// 等待機械復位完成
IF NOT xExecute THEN
	IF Cylinder.List.fbSameSizeCV_Block2.InRearPosition AND
	   Cylinder.List.fbTransmitCV_CamaraHoriz.InRearPosition AND
	   Motor.List.TransmitSameSideCV.InStopped THEN
		xComplete := TRUE;
	END_IF
ELSE
	IF Motor.List.TransmitSameSideCV.InStopped THEN
		xComplete := TRUE;
	END_IF
END_IF
END_METHOD

METHOD CyclicAction
VAR_INPUT
    itfTimingController : CBML.ITimingController;
END_VAR
VAR_OUTPUT
    xComplete : BOOL := TRUE;
    iErrorID : INT := 0;
END_VAR
VAR_INST
	bMoveConveyorBackward:BOOL;
END_VAR
xComplete := FALSE;
// Phase 2:寫請求,由 FB_MachineControl.A20_ConveyorArbitration 驅動 motor
IF __ISVALIDREF(SameSizeCVRequest) THEN
	SameSizeCVRequest.bCamera_NeedBackward := bMoveConveyorBackward;
END_IF

CASE uiCyclicStep OF
	0:	// 初始化
		bMoveConveyorBackward:=FALSE;
		uiCyclicStep :=1000;

	1000:	// 擋盒子 (Block2)
		TON_TimeOut.IN:=TRUE;
		Cylinder.List.fbSameSizeCV_Block2.M_Extend();
		Cylinder.List.fbTransmitCV_CamaraHoriz.M_Retract();
		IF Cylinder.List.fbSameSizeCV_Block2.InFrontPosition AND
			Cylinder.List.fbTransmitCV_CamaraHoriz.InRearPosition THEN
			TON_TimeOut.IN:=FALSE;
			uiCyclicStep :=1050;
		END_IF
		IF TON_TimeOut.Q THEN
			uiResumeStep := uiCyclicStep;
			iErrorID := 10;
		END_IF

	1050:	// 馬達反轉
		TON_ConveyorTimeOut.IN:=TRUE;
		bMoveConveyorBackward:=TRUE;
		Cylinder.List.fbSameSizeCV_Press1.M_Retract();
		IF Motor.List.TransmitSameSideCV.InBackWard AND
			Cylinder.List.fbSameSizeCV_Press1.InRearPosition THEN
			TON_ConveyorTimeOut.IN:= FALSE;
			uiCyclicStep :=1100;
		END_IF
		IF TON_ConveyorTimeOut.Q THEN
			uiResumeStep := uiCyclicStep;
			iErrorID := 10;
		END_IF

	1100:	// 檢查盒子到達擋塊 (Phase 2:撤銷 backward + 請求 HoldStill 拍照位)
		TON_ArriviedTimeOut.IN:=TRUE;
		TON_DelaySensor.IN:=Input.bSameSizeCV_BoxDetect2_Sensor;
		IF TON_DelaySensor.Q THEN
			TON_DelaySensor.IN :=FALSE;
			TON_ArriviedTimeOut.IN :=FALSE;
			Cylinder.List.fbSameSizeCV_Press1.M_Extend();
			bMoveConveyorBackward:=FALSE;
			IF __ISVALIDREF(SameSizeCVRequest) THEN
				SameSizeCVRequest.bCamera_NeedBackward := FALSE;
				SameSizeCVRequest.bCamera_HoldStill    := TRUE;	// 拍照位必須靜止
			END_IF
			uiCyclicStep :=1200;
		END_IF
		IF TON_ArriviedTimeOut.Q THEN
			uiResumeStep := uiCyclicStep;
			iErrorID := 9;
		END_IF

	1200:	// 發送拍照請求 & 壓住盒子
		TON_ConveyorTimeOut.IN:=TRUE;
		IF Cylinder.List.fbSameSizeCV_Press1.InFrontPosition AND
			Motor.List.TransmitSameSideCV.InStopped THEN
			TON_ConveyorTimeOut.IN:= FALSE;
			UseBoxCamera :=TRUE;
			uiCyclicStep :=1300;
		END_IF
		IF TON_ConveyorTimeOut.Q THEN
			uiResumeStep := uiCyclicStep;
			iErrorID := 10;
		END_IF

	1300:	// 等待 C# 拍照完成 (Camera 錯誤不可續做) — Phase 2:解 HoldStill,再次請求 backward
		TON_CameraTimeOut.IN:=TRUE;
		IF BoxCameraDone THEN
			TON_CameraTimeOut.IN :=FALSE;
			Cylinder.List.fbSameSizeCV_Block2.M_Retract();
			bMoveConveyorBackward:=TRUE;
			IF __ISVALIDREF(SameSizeCVRequest) THEN
				SameSizeCVRequest.bCamera_HoldStill := FALSE;
			END_IF
			uiCyclicStep :=1400;
		END_IF
		IF TON_CameraTimeOut.Q THEN
			uiResumeStep := uiCyclicStep;
			iErrorID := 11;
		END_IF

	1400:	// 盒子通過 Detect1 感測器
		TON_TimeOut.IN :=TRUE;
		IF Input.bSameSizeCV_BoxDetect3_Sensor THEN
			TON_TimeOut.IN :=FALSE;
			uiCyclicStep :=1500;
		END_IF
		IF TON_TimeOut.Q THEN
			uiResumeStep := uiCyclicStep;
			iErrorID := 12;
		END_IF

	1500:	// 離開感測器後撤銷 backward (Phase 2:arbiter 自動停)
		TON_DelaySensor.IN :=TRUE;
		IF NOT Input.bSameSizeCV_BoxDetect3_Sensor THEN
			TON_DelaySensor.IN :=FALSE;
			bMoveConveyorBackward:=FALSE;
			IF __ISVALIDREF(SameSizeCVRequest) THEN
				SameSizeCVRequest.bCamera_NeedBackward := FALSE;
			END_IF
			uiCyclicStep :=1600;
		END_IF
		IF TON_DelaySensor.Q THEN
			TON_DelaySensor.IN:=FALSE;
			bMoveConveyorBackward:=FALSE;
			IF __ISVALIDREF(SameSizeCVRequest) THEN
				SameSizeCVRequest.bCamera_NeedBackward := FALSE;
			END_IF
			uiCyclicStep :=1600;
		END_IF

	1600:	// 等待馬達停止
		IF Motor.List.TransmitSameSideCV.InStopped THEN
			xComplete :=TRUE;
		END_IF

END_CASE

IF TON_SameSizeBoxDetect1_Delay.Q THEN
	iErrorID := 13;
END_IF
END_METHOD

METHOD ExitAction
VAR_INPUT
    xAfterCleanup : BOOL;
    xInCopyCode : BOOL;
END_VAR
	uiCyclicStep    := 0;
	xAfterCleanup := true;
END_METHOD

METHOD M_GetErrorMsg : T_MaxString
VAR_INPUT
	xErrorID: INT;
END_VAR

VAR

END_VAR
CASE xErrorID OF
	1:
		M_GetErrorMsg := 'No Error';
	2:
		M_GetErrorMsg := 'FB_SameSizeCVCamera_Reverse ErrorID 2: Action time out';
	3:
		M_GetErrorMsg := 'FB_SameSizeCVCamera_Reverse ErrorID 3: Position Data invalid';
	4:
		M_GetErrorMsg := 'FB_SameSizeCVCamera_Reverse ErrorID 4: Block1 cylinder not ready';
	5:
		M_GetErrorMsg := 'FB_SameSizeCVCamera_Reverse ErrorID 5: Block2 cylinder not ready';
	6:
		M_GetErrorMsg := 'FB_SameSizeCVCamera_Reverse ErrorID 6: Press1 cylinder not ready';
	7:
		M_GetErrorMsg := 'FB_SameSizeCVCamera_Reverse ErrorID 7: Press2 cylinder not ready';
	8:
		M_GetErrorMsg := 'FB_SameSizeCVCamera_Reverse ErrorID 8: CameraHoriz cylinder not ready';
	9:
		M_GetErrorMsg :='FB_SameSizeCVCamera_Reverse ErrorID 9:  Box not arrived ';
	10:
		M_GetErrorMsg :='FB_SameSizeCVCamera_Reverse ErrorID 10: Cylinder timeout';
	11:
		M_GetErrorMsg :='FB_SameSizeCVCamera_Reverse ErrorID 11: C# BoxCameraDone timeout';
	12:
		M_GetErrorMsg :='FB_SameSizeCVCamera_Reverse ErrorID 12: Box cross sensor timeout';
	13:
		M_GetErrorMsg :='FB_SameSizeCVCamera_Reverse ErrorID 13: SameSizeConveyor full box infront ';
END_CASE
END_METHOD

METHOD ResetAction
VAR_OUTPUT
    xComplete : BOOL := TRUE;
END_VAR
xComplete := FALSE;

// ============================================================
// Resume 機制判斷
// ------------------------------------------------------------
// 當錯誤發生後，操作員可選擇：
//   1. 保持 xExecute = TRUE 並按 Reset → Resume (從錯誤點繼續)
//   2. 先關閉 xExecute，再重新啟動 → 從頭開始
// ============================================================
bResumeEnabled := xExecute;

// 如果不是 Resume 模式，清除 Resume 步驟記錄
IF NOT bResumeEnabled THEN
	uiResumeStep := 0;
END_IF

// 清除所有 Timer
TON_DelaySensor.IN 		:= FALSE;
TON_TimeOut.IN 			:= FALSE;
TON_ArriviedTimeOut.IN 	:= FALSE;
TON_CameraTimeOut.IN 	:= FALSE;
TON_ConveyorTimeOut.IN 	:= FALSE;

xComplete := TRUE;
END_METHOD

METHOD StartAction
VAR_OUTPUT
    xComplete : BOOL := TRUE;
	iErrorID : INT := 0;
END_VAR
VAR
	bIsResumeMode : BOOL;	// 局部變數：記錄是否為 Resume 模式
END_VAR
xComplete := FALSE;

// 清除所有 Timer
TON_DelaySensor.IN 		:= FALSE;
TON_TimeOut.IN 			:= FALSE;
TON_ArriviedTimeOut.IN 	:= FALSE;
TON_CameraTimeOut.IN 	:= FALSE;
TON_ConveyorTimeOut.IN 	:= FALSE;

// ============================================================
// Resume 機制處理
// ------------------------------------------------------------
// 可 Resume 的錯誤: 氣缸/馬達/等待盒子
// 不可 Resume 的錯誤: Step 1300 (C# 拍照失敗)
// ============================================================
bIsResumeMode := bResumeEnabled AND uiResumeStep > 0 AND uiResumeStep <> 1300;

IF bResumeEnabled AND uiResumeStep > 0 THEN
	IF uiResumeStep = 1300 THEN
		// Camera 錯誤：不可 Resume，強制從頭開始
		uiCyclicStep 	:= 0;
		UseBoxCamera 	:= FALSE;
		BoxCameraDone 	:= FALSE;
	ELSE
		// 其他錯誤：允許 Resume (人工已確認可繼續)
		uiCyclicStep := uiResumeStep;
	END_IF
	// 清除 Resume 旗標
	bResumeEnabled 	:= FALSE;
	uiResumeStep 	:= 0;
ELSE
	// 正常模式：從頭開始
	uiCyclicStep 	:= 0;
	UseBoxCamera 	:= FALSE;
	BoxCameraDone 	:= FALSE;
END_IF

// ============================================================
// 啟動前錯誤檢查
// ============================================================
IF TON_SameSizeBoxDetect1_Delay.Q THEN
	iErrorID := 13;
END_IF

IF Cylinder.List.fbSameSizeCV_Block1.xError THEN
	iErrorID := 4;
END_IF
IF Cylinder.List.fbSameSizeCV_Block2.xError THEN
	iErrorID := 5;
END_IF
IF Cylinder.List.fbSameSizeCV_Press1.xError THEN
	iErrorID := 6;
END_IF
IF Cylinder.List.fbSameSizeCV_Press2.xError THEN
	iErrorID := 7;
END_IF
IF Cylinder.List.fbTransmitCV_CamaraHoriz.xError THEN
	iErrorID := 8;
END_IF
IF Motor.List.TransmitSameSideCV.xError THEN
	iErrorID := 9;
END_IF

// 完成條件：Resume 模式直接完成，正常模式需檢查初始位置
IF bIsResumeMode OR
   (Cylinder.List.fbSameSizeCV_Block2.InRearPosition AND
    Motor.List.TransmitSameSideCV.InStopped) THEN
	xComplete := TRUE;
END_IF
END_METHOD

END_FUNCTION_BLOCK

// ---- Library/20_MachineUnits/22_AllocateArea/Service/FB_DifferentCVCamera.TcPOU
FUNCTION_BLOCK FB_DifferentCVCamera EXTENDS FB_ActionBasic
VAR_INPUT
    xExecute    : BOOL;
    xAbort      : BOOL;
	xReset		: BOOL;
    Cylinder 	: REFERENCE TO UNI_CylinderList;
    TimeOut  	: LREAL := 600; // Unit : s
	Input		: ST_InputTable;
	OutPut		: ST_OutputTable;
	Motor		: REFERENCE TO UNI_MotorList;
	BoxCameraDone :BOOL;
END_VAR	
VAR_OUTPUT
    xAborted : BOOL;
    iErrorID : INT;
    ErrorMsg : STRING;
	UseBoxCamera	:BOOL;
END_VAR
VAR
    StateBehaviour   : CBML.ETrigATo;
    CurrentPosition : ST_PositionTable;
	uiCyclicStep    : UINT := 0;
	TON_DelaySensor	:TON;
	TON_TimeOut		:TON;
	TON_ArriviedTimeOut :TON ;
	TON_CameraTimeOut	:TON;
	TON_ConveyorTimeOut	:TON;
	Reset_Rtrig 	:R_TRIG;
	fbExecuteEdgeDetect :FB_EdgeDetect;
	// ========== Resume 續做機制 ==========
	uiResumeStep	: UINT := 0;		// 錯誤發生時記錄的步驟，供續做使用
	bResumeEnabled	: BOOL := FALSE;	// 續做模式啟用旗標
END_VAR

THIS^.IBehaviourModel := StateBehaviour;
StateBehaviour(xExecute := xExecute,
              xAbort := xAbort OR fbExecuteEdgeDetect.xFallingEdge,
              udiTimeOut := LREAL_TO_UDINT( TimeOut*1000000),
              xDone => xDone,
              xBusy => xBusy,
              xError => xError,
              xAborted => xAborted);

iErrorID := StateBehaviour._model.iErrorID;
ErrorMsg := M_GetErrorMsg(xErrorID := iErrorID);

fbExecuteEdgeDetect(xInput :=xExecute);

Reset_Rtrig(CLK:= xReset);
IF Reset_Rtrig.Q THEN
	StateBehaviour.ResetModel(xCommit:=xReset);
END_IF

A00_BaseUnits();

ACTION A00_BaseUnits:
TON_DelaySensor(PT:= T#1S);
TON_TimeOut(PT := T#20S);
TON_ArriviedTimeOut(PT:= T#60S);
TON_CameraTimeOut(PT :=T#250S);
TON_ConveyorTimeOut(PT :=T#60S);
END_ACTION

METHOD CleanupAction
VAR_INPUT
    xAbortProposed : BOOL;
    iErrorIDProposed: INT;
END_VAR
VAR_OUTPUT
    xComplete : BOOL := TRUE;
    xAbort: BOOL := xAbortProposed;
 	iErrorID : INT := iErrorIDProposed;
END_VAR
xComplete := FALSE;

// ============================================================
// Resume 機制：保存當前步驟供後續 Resume 使用
// ============================================================
IF uiResumeStep = 0 THEN
	uiResumeStep := uiCyclicStep;
END_IF

// 清除所有 Timer
TON_DelaySensor.IN 		:= FALSE;
TON_TimeOut.IN 			:= FALSE;
TON_ArriviedTimeOut.IN 	:= FALSE;
TON_CameraTimeOut.IN 	:= FALSE;
TON_ConveyorTimeOut.IN 	:= FALSE;

// 重置輸出信號
UseBoxCamera 	:= FALSE;
BoxCameraDone 	:= FALSE;

// 機械復位到安全狀態
IF NOT xExecute THEN 
	Cylinder.List.fbDifferentSizeCV_Block1.M_Retract();
END_IF
Motor.List.TransmitDifferentSideCV.M_MotorStop();

// 等待機械復位完成
IF NOT xExecute THEN
	IF Cylinder.List.fbDifferentSizeCV_Block1.InRearPosition AND
	   Motor.List.TransmitDifferentSideCV.InStopped THEN
		xComplete := TRUE;
	END_IF
ELSE	
	IF Motor.List.TransmitDifferentSideCV.InStopped THEN
		xComplete := TRUE;
	END_IF
END_IF
END_METHOD

METHOD CyclicAction
VAR_INPUT
    itfTimingController : CBML.ITimingController;
END_VAR
VAR_OUTPUT
    xComplete : BOOL := TRUE;
    iErrorID : INT := 0;
END_VAR
VAR_INST
	bMoveConveyorForward	 : BOOL;
END_VAR
xComplete := FALSE;
IF bMoveConveyorForward THEN
	IF NOT Motor.List.TransmitDifferentSideCV.InBackWard THEN
		Motor.List.TransmitDifferentSideCV.M_MoveForward();
	END_IF
END_IF
CASE uiCyclicStep OF
	0:	// 初始化
		bMoveConveyorForward:=FALSE;
		uiCyclicStep :=1000;
		
	1000:	// 擋第一個盒子
		TON_TimeOut.IN:=TRUE;
		Cylinder.List.fbDifferentSizeCV_Block1.M_Extend();
		Cylinder.List.fbTransmitCV_CamaraHoriz.M_Extend();
		IF Cylinder.List.fbDifferentSizeCV_Block1.InFrontPosition AND
			Cylinder.List.fbTransmitCV_CamaraHoriz.InFrontPosition THEN
			TON_TimeOut.IN:=FALSE;
			uiCyclicStep :=1050;
		END_IF
		IF TON_TimeOut.Q THEN
			uiResumeStep := uiCyclicStep;
			iErrorID := 7;
		END_IF

	1050:	// 馬達前進
		TON_ConveyorTimeOut.IN:=TRUE;
		bMoveConveyorForward:=TRUE;
		Cylinder.List.fbDifferentSizeCV_Press1.M_Retract();
		IF Motor.List.TransmitDifferentSideCV.InForWard AND
			Cylinder.List.fbDifferentSizeCV_Press1.InRearPosition THEN
			TON_ConveyorTimeOut.IN:= FALSE;
			uiCyclicStep :=1100;
		END_IF
		IF TON_ConveyorTimeOut.Q THEN
			uiResumeStep := uiCyclicStep;
			iErrorID := 7;
		END_IF

	1100:	// 檢查盒子到達擋塊
		TON_ArriviedTimeOut.IN:=TRUE;
		TON_DelaySensor.IN:=Input.bDifferentSizeCV_BoxDetect2_Sensor;
		IF TON_DelaySensor.Q THEN
			TON_DelaySensor.IN :=FALSE;
			TON_ArriviedTimeOut.IN :=FALSE;
			Cylinder.List.fbDifferentSizeCV_Press1.M_Extend();
			bMoveConveyorForward:=FALSE;
			Motor.List.TransmitDifferentSideCV.M_MotorStop();
			uiCyclicStep :=1200;
		END_IF
		IF TON_ArriviedTimeOut.Q THEN
			uiResumeStep := uiCyclicStep;
			iErrorID := 8;
		END_IF

	1200:	// 發送拍照請求 & 擋住第二個盒子
		TON_ConveyorTimeOut.IN:=TRUE;
		IF Cylinder.List.fbDifferentSizeCV_Press1.InFrontPosition AND
			Motor.List.TransmitDifferentSideCV.InStopped THEN
			TON_ConveyorTimeOut.IN:= FALSE;
			UseBoxCamera :=TRUE;
			uiCyclicStep :=1300;
		END_IF
		IF TON_ConveyorTimeOut.Q THEN
			uiResumeStep := uiCyclicStep;
			iErrorID := 9;
		END_IF

	1300:	// 等待 C# 拍照完成 (Camera 錯誤不可續做)
		TON_CameraTimeOut.IN:=TRUE;
		IF BoxCameraDone THEN
			TON_CameraTimeOut.IN :=FALSE;
			Cylinder.List.fbDifferentSizeCV_Block1.M_Retract();
			bMoveConveyorForward:=TRUE;
			uiCyclicStep :=1400;
		END_IF
		IF TON_CameraTimeOut.Q THEN
			uiResumeStep := uiCyclicStep;
			iErrorID :=10;
		END_IF

	1400:	// 盒子通過 Detect1 感測器
		TON_TimeOut.IN :=TRUE;
		IF Input.bDifferentSizeCV_BoxDetect1_Sensor THEN
			TON_TimeOut.IN :=FALSE;
			uiCyclicStep :=1500;
		END_IF
		IF TON_TimeOut.Q THEN
			uiResumeStep := uiCyclicStep;
			iErrorID :=11;
		END_IF

	1500:	// 離開感測器後停止馬達
		TON_DelaySensor.IN:=TRUE;
		IF NOT Input.bDifferentSizeCV_BoxDetect1_Sensor THEN
			TON_DelaySensor.IN:=FALSE;
			bMoveConveyorForward:=FALSE;
			Motor.List.TransmitDifferentSideCV.M_MotorStop();
			uiCyclicStep :=1600;
		END_IF
		IF TON_DelaySensor.Q THEN
			TON_DelaySensor.IN:=FALSE;
			bMoveConveyorForward:=FALSE;
			Motor.List.TransmitDifferentSideCV.M_MotorStop();
			uiCyclicStep :=1600;
		END_IF
	
	1600:	// 等待馬達停止
		IF Motor.List.TransmitDifferentSideCV.InStopped THEN
			xComplete :=TRUE;
		END_IF

END_CASE
END_METHOD

METHOD ExitAction
VAR_INPUT
    xAfterCleanup : BOOL;
    xInCopyCode : BOOL;
END_VAR
END_METHOD

METHOD M_GetErrorMsg : T_MaxString
VAR_INPUT
	xErrorID: INT;
END_VAR

VAR
	
END_VAR
CASE xErrorID OF
	0:
		M_GetErrorMsg := 'No Error';
	1:
		M_GetErrorMsg := 'FB_DifferentCVCamera ErrorID 1: Action time out';
	2:
		M_GetErrorMsg := 'FB_DifferentCVCamera ErrorID 2: Position Data invalid';
	3:
		M_GetErrorMsg := 'FB_DifferentCVCamera ErrorID 3: Block1 cylinder not ready';
	4:
		M_GetErrorMsg := 'FB_DifferentCVCamera ErrorID 4: Press1 cylinder not ready';
	5:
		M_GetErrorMsg := 'FB_DifferentCVCamera ErrorID 5: CamaraHoriz cylinder not ready';
	6:
		M_GetErrorMsg := 'FB_DifferentCVCamera ErrorID 6: DifferentCV not ready ';
	7:
		M_GetErrorMsg := 'FB_DifferentCVCamera ErrorID 7: Cylinder timeout';
	8:
		M_GetErrorMsg :='FB_DifferentCVCamera ErrorID 8: photo area have not box timeout';
	9:
		M_GetErrorMsg :='FB_DifferentCVCamera ErrorID 9: motor & cylinder timeout';
	10:
		M_GetErrorMsg :='FB_DifferentCVCamera ErrorID 10: C# BoxCameraDone timeout';
	11:
		M_GetErrorMsg :='FB_DifferentCVCamera ErrorID 11: Box cross sensor not detact timeout';
		
	20:
		M_GetErrorMsg :='FB_DifferentCVCamera ErrorID 20: Differnet conveyor full box infront';
END_CASE
END_METHOD

METHOD ResetAction
VAR_OUTPUT
    xComplete : BOOL := TRUE;
END_VAR
xComplete := FALSE;

// ============================================================
// Resume 機制判斷
// ------------------------------------------------------------
// 當錯誤發生後，操作員可選擇：
//   1. 保持 xExecute = TRUE 並按 Reset → Resume (從錯誤點繼續)
//   2. 先關閉 xExecute，再重新啟動 → 從頭開始
// ============================================================
bResumeEnabled := xExecute;

// 如果不是 Resume 模式，清除 Resume 步驟記錄
IF NOT bResumeEnabled THEN
	uiResumeStep := 0;
END_IF

// 清除所有 Timer
TON_DelaySensor.IN 		:= FALSE;
TON_TimeOut.IN 			:= FALSE;
TON_ArriviedTimeOut.IN 	:= FALSE;
TON_CameraTimeOut.IN 	:= FALSE;
TON_ConveyorTimeOut.IN 	:= FALSE;

xComplete := TRUE;
END_METHOD

METHOD StartAction
VAR_OUTPUT
    xComplete : BOOL := TRUE;
	iErrorID : INT := 0;
END_VAR
VAR
	bIsResumeMode : BOOL;	// 局部變數：記錄是否為 Resume 模式
END_VAR
xComplete := FALSE;

// 清除所有 Timer
TON_DelaySensor.IN 		:= FALSE;
TON_TimeOut.IN 			:= FALSE;
TON_ArriviedTimeOut.IN 	:= FALSE;
TON_CameraTimeOut.IN 	:= FALSE;
TON_ConveyorTimeOut.IN 	:= FALSE;

// ============================================================
// Resume 機制處理
// ------------------------------------------------------------
// 可 Resume 的錯誤: Error 7, 8, 9, 11 (氣缸/馬達/等待盒子)
// 不可 Resume 的錯誤: Error 10 (C# 拍照失敗), Error 20 (輸送帶滿載)
// ============================================================
bIsResumeMode := bResumeEnabled AND uiResumeStep > 0 AND uiResumeStep <> 1300;

IF bResumeEnabled AND uiResumeStep > 0 THEN
	IF uiResumeStep = 1300 THEN
		// Camera 錯誤：不可 Resume，強制從頭開始
		uiCyclicStep 	:= 0;
		UseBoxCamera 	:= FALSE;
		BoxCameraDone 	:= FALSE;
	ELSE
		// 其他錯誤：允許 Resume (人工已確認可繼續)
		uiCyclicStep := uiResumeStep;
	END_IF
	// 清除 Resume 旗標
	bResumeEnabled 	:= FALSE;
	uiResumeStep 	:= 0;
ELSE
	// 正常模式：從頭開始
	uiCyclicStep 	:= 0;
	UseBoxCamera 	:= FALSE;
	BoxCameraDone 	:= FALSE;
END_IF

// ============================================================
// 啟動前錯誤檢查
// ============================================================
IF Input.bDifferentSizeCV_BoxDetect1_Sensor THEN
	iErrorID := 20;
END_IF

IF Cylinder.List.fbDifferentSizeCV_Block1.xError THEN
	iErrorID := 3;
END_IF
IF Cylinder.List.fbDifferentSizeCV_Press1.xError THEN
	iErrorID := 4;
END_IF
IF Cylinder.List.fbTransmitCV_CamaraHoriz.xError THEN
	iErrorID := 5;
END_IF
IF Motor.List.TransmitDifferentSideCV.xError THEN
	iErrorID := 6;
END_IF

// 完成條件：Resume 模式直接完成，正常模式需檢查初始位置
IF bIsResumeMode OR
   (Cylinder.List.fbDifferentSizeCV_Block1.InRearPosition AND
    Motor.List.TransmitDifferentSideCV.InStopped) THEN
	xComplete := TRUE;
END_IF
END_METHOD

END_FUNCTION_BLOCK

// ---- Library/20_MachineUnits/22_AllocateArea/Service/FB_SameSizeCV_ReverseBatchPickAndPhoto.TcPOU
// FB_SameSizeCV_ReverseBatchPickAndPhoto
// 逆向拍照批次入料服務
// Pipeline 三軌平行:
//   Track 1 (小手臂): 從鐵盤取盒放到同尺寸軌道 (ShippingRobotTransfer)
//   Track 2 (拍照):   觸發逆向拍照, 接收 C# 回傳結果
//   Track 3 (大手臂): 雙爪/單爪搬運到倉庫或 NG 區 (倉儲 Fanuc Robot)
//
// 狀態機架構: FB_ObjectBase_V2 + IBasicElement
//   DORMANT → EXECUTING → DONE / ABORTING → ABORTED → RESETTING → DORMANT
//
// Handshake: 由 FB_AllocateAreaWithRoundbelt 逐欄位 link ADS 結構

FUNCTION_BLOCK FB_SameSizeCV_ReverseBatchPickAndPhoto EXTENDS FB_ObjectBase_V2 IMPLEMENTS IBasicElement

VAR_INPUT
	// ===== 鐵盤 Sensor (C# → PLC, 目前 C# 模擬，後續改硬體訊號) =====
	bLeftPlateReady		: BOOL;
	bRightPlateReady	: BOOL;

	// ===== 鐵盤配置 (C# → PLC) =====
	LeftPlate			: ARRAY[0..3] OF BOOL;
	RightPlate			: ARRAY[0..3] OF BOOL;
	bLeftConfigReady	: BOOL;
	bRightConfigReady	: BOOL;

	// ===== 拍照結果 (C# → PLC) =====
	BoxCameraDone		: BOOL;
	CameraIsOK			: BOOL;
	CameraWarehouse		: INT;
	CameraLevel			: INT;
	CameraTrack			: INT;

	// ===== 硬體 REFERENCE =====
	Cylinder			: REFERENCE TO UNI_CylinderList;
	Motor				: REFERENCE TO UNI_MotorList;
	SameSizeCVRequest	: REFERENCE TO ST_SameSizeCVRequest;	// Phase 2 仲裁,傳到 3 個 sub-FB
	Input				: ST_InputTable;
	OutPut				: ST_OutputTable;
	StorageRobot		: REFERENCE TO FB_FanucRobot_Basic_V2;
	ShippingRobot		: REFERENCE TO FB_FanucRobot_Basic_V2;
	WareHouse			: REFERENCE TO FB_WareHouse;
	
	Stop				: BOOL;

	// ===== 設定 =====
	PlateWaitTimeout	: TIME := T#60S;
	WaitPairTimeout		: TIME := T#15S;
	BatchTimeout		: TIME := T#600S;
END_VAR

VAR_OUTPUT
	// ===== 鐵盤狀態 (PLC → C#) =====
	bLeftPlateArrived	: BOOL;
	bRightPlateArrived	: BOOL;
	bLeftPlateDone		: BOOL;
	bRightPlateDone		: BOOL;

	// ===== 拍照請求 (PLC → C#) =====
	UseBoxCamera		: BOOL;

	// ===== 狀態監控 (PLC → C#) =====
	uiUnphotographedCount	: UINT;
	uiTotalProcessed		: UINT;
	uiTransportedCount		: UINT;
	
	
END_VAR

VAR
	strStatus			: STRING;
	_UniqueErrorCode	: STRING;
	_bRetry				: BOOL;

	// ===== Track 1: 小手臂取盒 =====
	uiPickStep				: UINT := 0;
	uiCurrentSide			: UINT := 0;		// 0=Left, 1=Right
	uiCurrentSlot			: UINT := 0;		// 0..3
	bPickTrackDone			: BOOL;
	bLeftProcessed			: BOOL;
	bRightProcessed			: BOOL;
	bLeftPlateReady_Prev	: BOOL;
	bRightPlateReady_Prev	: BOOL;
	bLeftConfigLatched		: BOOL;
	bRightConfigLatched		: BOOL;
	bLeftConfigReady_Prev	: BOOL;
	bRightConfigReady_Prev	: BOOL;

	// ===== Track 2: 拍照 =====
	uiCameraStep			: UINT := 0;
	uiCameraRequestCount	: UINT := 0;

	// ===== Track 3: 大手臂搬運 =====
	uiTransportStep		: UINT := 0;
	BoxQueue			: ST_ReverseBatchBoxQueue;
	stGripA				: ST_ReverseBatchBoxResult;
	stGripB				: ST_ReverseBatchBoxResult;
	bUseDualGrip		: BOOL;
	bTransportBusy		: BOOL;

	// ===== Timers =====
	tonTimeOut				: TON;
	TON_PlateWaitTimeout	: TON;
	TON_PickupTimeout		: TON;
	TON_CameraTimeout		: TON;
	TON_ConfigTimeout		: TON;
	TON_WaitPairTimeout		: TON;
	TON_CameraClearTimeout	: TON;

	// ===== Resume =====
	uiResumePickStep		: UINT := 0;
	uiResumeCameraStep		: UINT := 0;
	uiResumeTransportStep	: UINT := 0;
	
	// 內部使用Service
	ShippingTransfer	: FB_ShippingRobotTransfer;
	BoxToWareHouse		: FB_SameSizeCV_ReverseBoxToWareHouse;
	_fbSameSizeCV_ReverseCamera	: FB_SameSizeCVCamera_Reverse;
END_VAR

SUPER^.A10_StateControl();
A00_BasicUnits();

ACTION A00_BasicUnits:
tonTimeOut(PT := BatchTimeout);
TON_PlateWaitTimeout(PT := PlateWaitTimeout);
TON_PickupTimeout(PT := T#60S);
TON_CameraTimeout(PT := T#600S);
TON_ConfigTimeout(PT := T#60S);
TON_WaitPairTimeout(PT := WaitPairTimeout);
TON_CameraClearTimeout(PT := T#30S);


ShippingTransfer(
	Execute:= , 
	Abort:= , 
	Reset:= , 
	Pause:= , 
	ObjectName:= , 
	Busy=> , 
	Done=> , 
	Aborted=> , 
	Error=> , 
	Paused=> , 
	ErrorID=> , 
	Status=> , 
	UniqueErrorCode=> , 
	Robot:= ShippingRobot,
	Info:= ,
	Stop:= Stop,
	Input:= INPUT,
	Output:= OUTPUT,
	Motor:= Motor,
	SameSizeCVRequest:= SameSizeCVRequest,
	Cylinder:= Cylinder,
	Buzz:= ,
	RedLamp:= , 
	bCompleteRequest:= , 
	fbShippingHomingBusy:= , 
	bTransCVInPosition_Left=> , 
	bTransCVInPosition_Right=> );
	
BoxToWareHouse(
	Execute:= , 
	Abort:= , 
	Reset:= , 
	Pause:= , 
	ObjectName:= , 
	Busy=> , 
	Done=> , 
	Aborted=> , 
	Error=> , 
	Paused=> , 
	ErrorID=> , 
	Status=> , 
	UniqueErrorCode=> , 
	bBoxA_Enable:= ,
	eBoxA_Destination:= ,
	iBoxA_Warehouse:= ,
	iBoxA_Level:= ,
	iBoxA_Track:= ,
	iBoxA_PullOutSide:= ,
	bBoxB_Enable:= ,
	eBoxB_Destination:= ,
	iBoxB_Warehouse:= ,
	iBoxB_Level:= ,
	iBoxB_Track:= ,
	iBoxB_PullOutSide:= ,
	NGAreaPosition:= ,
	PickupPosition:= ,
	Cylinder:= Cylinder,
	Motor:= Motor,
	SameSizeCVRequest:= SameSizeCVRequest,
	Input:= Input,
	OutPut:= OutPut,
	StorageRobot:= StorageRobot,
	WareHouse:= WareHouse,
	PullOutConveyor:= ,
	Stop:= Stop,
	bBoxA_Done=> ,
	bBoxB_Done=> );
	
_fbSameSizeCV_ReverseCamera(
	xDone=> , 
	xBusy=> , 
	xError=> , 
	xExecute:= , 
	xAbort:= , 
	xReset:= , 
	Cylinder:= Cylinder,
	TimeOut:= ,
	Input:= input,
	OutPut:= output,
	Motor:= Motor,
	SameSizeCVRequest:= SameSizeCVRequest,
	BoxCameraDone:= ,
	xAborted=> , 
	iErrorID=> , 
	ErrorMsg=> , 
	UseBoxCamera=> );
END_ACTION

METHOD M_GetErrorMsg : T_MaxString
VAR_INPUT
END_VAR
IF _UniqueErrorCode = 'E_PICKUP_TIMEOUT' THEN
	M_GetErrorMsg := 'FB_SameSizeCV_ReverseBatchPickAndPhoto: ShippingRobot pickup timeout';
ELSIF _UniqueErrorCode = 'E_BIGARM_TIMEOUT' THEN
	M_GetErrorMsg := 'FB_SameSizeCV_ReverseBatchPickAndPhoto: BigArm transport timeout';
ELSIF _UniqueErrorCode = 'E_CONVEYOR_FULL' THEN
	M_GetErrorMsg := 'FB_SameSizeCV_ReverseBatchPickAndPhoto: Conveyor full (queue overflow)';
ELSIF _UniqueErrorCode = 'E_CONFIG_TIMEOUT' THEN
	M_GetErrorMsg := 'FB_SameSizeCV_ReverseBatchPickAndPhoto: Waiting C# plate config timeout';
ELSIF _UniqueErrorCode = 'E_CAMERA_TIMEOUT' THEN
	M_GetErrorMsg := 'FB_SameSizeCV_ReverseBatchPickAndPhoto: Camera timeout';
ELSIF _UniqueErrorCode = 'E_CAMERA_CLEAR_TIMEOUT' THEN
	M_GetErrorMsg := 'FB_SameSizeCV_ReverseBatchPickAndPhoto: C# did not clear BoxCameraDone';
ELSIF _UniqueErrorCode = 'E_BATCH_TIMEOUT' THEN
	M_GetErrorMsg := 'FB_SameSizeCV_ReverseBatchPickAndPhoto: Batch global timeout';
ELSIF _UniqueErrorCode = '' THEN
	M_GetErrorMsg := 'No Error';
ELSE
	M_GetErrorMsg := _UniqueErrorCode;
END_IF
END_METHOD

// 已中止狀態 — 等待 Reset 信號，支援 Resume
METHOD M_STATE_ABORTED
VAR_INPUT
END_VAR
IF NOT _bRetry THEN
	Busy 			:= FALSE;
	Aborted 		:= TRUE;
	Error 			:= TRUE;
	Status 			:= strStatus;
	uiAbortingStep 	:= 0;
	_AbortCompleted := FALSE;
END_IF


IF reset THEN
	_bRetry := TRUE;
	Aborted := FALSE;
	Error 	:= FALSE;	
END_IF

IF NOT Execute THEN
	eState := STATE_RESETTING;
END_IF

// 等待外部 Reset → 恢復或重置
IF Execute
	AND _bRetry 
	AND NOT StorageRobot._DI1.Error 
	AND NOT ShippingRobot._DI1.Error 
	AND NOT StorageRobot.Halt
	AND NOT StorageRobot.Halt
THEN
	status := 'FB_SameSizeCV_ReverseBatchPickAndPhoto: Retry Complete';
	// 恢復三軌步驟
	uiPickStep := uiResumePickStep;
	uiCameraStep := uiResumeCameraStep;
	uiTransportStep := uiResumeTransportStep;
	uiResumePickStep := 0;
	uiResumeCameraStep := 0;
	uiResumeTransportStep := 0;
	// 跳過初始化，直接進入三軌運行
	uiExecutingStep := 100;

	eState := STATE_RESETTING;
END_IF
END_METHOD

// 中止狀態 — 停止所有 Track，保存 Resume 步驟
METHOD M_STATE_ABORTING
VAR_INPUT
END_VAR
CASE uiAbortingStep OF
0:
	// 保存所有 Track Resume 步驟 (如果尚未保存)
	IF uiResumePickStep = 0 AND uiResumeTransportStep = 0 AND uiResumeCameraStep = 0 THEN
		uiResumePickStep := uiPickStep;
		uiResumeCameraStep := uiCameraStep;
		uiResumeTransportStep := uiTransportStep;
	END_IF

	// 清除所有 Timer
	tonTimeOut.IN				:= FALSE;
	TON_PlateWaitTimeout.IN		:= FALSE;
	TON_PickupTimeout.IN		:= FALSE;
	TON_CameraTimeout.IN		:= FALSE;
	TON_ConfigTimeout.IN		:= FALSE;
	TON_WaitPairTimeout.IN		:= FALSE;
	TON_CameraClearTimeout.IN	:= FALSE;

	// 清除輸出
	UseBoxCamera := FALSE;

	// 停止小手臂
	ShippingTransfer.Execute := FALSE;
	ShippingTransfer.Abort := TRUE;

	// 停止大手臂子服務
	BoxToWareHouse.Execute := FALSE;
	BoxToWareHouse.Abort := TRUE;

	uiAbortingStep := 100;

100:
	// 等待子服務停止 (ShippingTransfer + BoxToWareHouse)
	IF (NOT ShippingTransfer.Busy OR ShippingTransfer.Aborted)
	   AND (NOT BoxToWareHouse.Busy OR BoxToWareHouse.Aborted) THEN
		ShippingTransfer.Abort := FALSE;
		BoxToWareHouse.Abort := FALSE;
		uiAbortingStep := 9999;
	END_IF

9999:
	_AbortCompleted := TRUE;
END_CASE

IF NOT Execute THEN
	eState := STATE_RESETTING;
ELSIF _AbortCompleted THEN
	eState := STATE_Aborted;
END_IF
END_METHOD

METHOD M_STATE_DONE
VAR_INPUT
END_VAR
Busy := FALSE;
Done := TRUE;
tonTimeOut.IN := FALSE;

// 等待外部取消 Execute 後進入 RESETTING
IF NOT Execute THEN
	eState := STATE_RESETTING;
END_IF
END_METHOD

METHOD M_STATE_DORMANT
VAR_INPUT
END_VAR
VAR
	i : UINT;
END_VAR
// 清除所有輸出與內部狀態
Busy				:= FALSE;
Done				:= FALSE;
Aborted				:= FALSE;
Error				:= FALSE;
ErrorID				:= 0;
Status				:= '';
_ResetCompleted		:= FALSE;
_Error				:= FALSE;
_Executed			:= FALSE;
_Abort				:= FALSE;
uiExecutingStep		:= 0;
uiResettingStep		:= 0;
uiAbortingStep		:= 0;

tonTimeOut.IN		:= FALSE;
_UniqueErrorCode	:= '';
_bRetry				:= FALSE;

// 清除 Track 變數
uiPickStep 			:= 0;
uiCameraStep 		:= 0;
uiTransportStep 	:= 0;
uiCameraRequestCount := 0;
uiUnphotographedCount := 0;
uiTotalProcessed 	:= 0;
uiTransportedCount 	:= 0;
bPickTrackDone 		:= FALSE;
bLeftProcessed 		:= FALSE;
bRightProcessed 	:= FALSE;
bTransportBusy 		:= FALSE;
bUseDualGrip 		:= FALSE;
UseBoxCamera 		:= FALSE;
bLeftPlateArrived 	:= FALSE;
bRightPlateArrived 	:= FALSE;
bLeftPlateDone 		:= FALSE;
bRightPlateDone 	:= FALSE;
bLeftPlateReady_Prev := FALSE;
bRightPlateReady_Prev := FALSE;
bLeftConfigLatched 	:= FALSE;
bRightConfigLatched := FALSE;
bLeftConfigReady_Prev := FALSE;
bRightConfigReady_Prev := FALSE;

uiResumePickStep 	:= 0;
uiResumeCameraStep 	:= 0;
uiResumeTransportStep := 0;

// 清除 Timers
TON_PlateWaitTimeout.IN		:= FALSE;
TON_PickupTimeout.IN		:= FALSE;
TON_CameraTimeout.IN		:= FALSE;
TON_ConfigTimeout.IN		:= FALSE;
TON_WaitPairTimeout.IN		:= FALSE;
TON_CameraClearTimeout.IN	:= FALSE;

// 清除佇列
BoxQueue.WriteIdx 	:= 0;
BoxQueue.ReadIdx 	:= 0;
BoxQueue.Count 		:= 0;
FOR i := 0 TO 15 DO
	BoxQueue.Boxes[i].bActive := FALSE;
END_FOR
stGripA.bActive := FALSE;
stGripB.bActive := FALSE;

_AbortCompleted := FALSE;

// 監聽外部 Execute/Reset (由 FB_AllocateAreaWithRoundbelt link ADS)
IF Execute AND NOT Stop THEN
	eState := STATE_EXECUTING;
END_IF
END_METHOD

METHOD M_STATE_ERROR
VAR_INPUT
END_VAR
Busy := FALSE;
Error := TRUE;
Status := strStatus;
tonTimeOut.IN := FALSE;

IF NOT Execute THEN
	eState := STATE_RESETTING;
END_IF
END_METHOD

// 執行主狀態 — Pipeline 三軌平行
// ═══════════════════════════════════════════════════
// uiExecutingStep:
//   0:   初始化 (清除計數/佇列)
//   100: 三軌平行運行 + Done 判斷
// ═══════════════════════════════════════════════════
METHOD M_STATE_EXECUTING
VAR_INPUT
END_VAR
Busy := TRUE;
tonTimeOut.IN := TRUE;

// 外部中止 (由 FB_AllocateAreaWithRoundbelt 傳入 Abort)
IF Abort THEN
	strStatus := 'FB_SameSizeCV_ReverseBatchPickAndPhoto: Aborted';
	_UniqueErrorCode := 'E_ABORT';
	_Abort := TRUE;
	RETURN;
END_IF

// 批次全域逾時
IF tonTimeOut.Q THEN
	strStatus := 'FB_SameSizeCV_ReverseBatchPickAndPhoto: Batch timeout';
	_UniqueErrorCode := 'E_BATCH_TIMEOUT';
	// 保存所有 Track 的 Resume 步驟
	uiResumePickStep := uiPickStep;
	uiResumeCameraStep := uiCameraStep;
	uiResumeTransportStep := uiTransportStep;
	_Abort := TRUE;
	RETURN;
END_IF

// Stop 時暫停所有 Timeout (含批次全域逾時)
IF Stop THEN
	tonTimeOut.IN             := FALSE;
	TON_PickupTimeout.IN      := FALSE;
	TON_CameraTimeout.IN      := FALSE;
	TON_ConfigTimeout.IN      := FALSE;
	TON_WaitPairTimeout.IN    := FALSE;
	TON_CameraClearTimeout.IN := FALSE;
END_IF

CASE uiExecutingStep OF

// ═══════════════════════════════════════════════════
// Step 0: 初始化
// ═══════════════════════════════════════════════════
0:
	uiPickStep := 0;
	uiCameraStep := 0;
	uiTransportStep := 0;
	uiCameraRequestCount := 0;
	uiUnphotographedCount := 0;
	uiTotalProcessed := 0;
	uiTransportedCount := 0;
	bPickTrackDone := FALSE;
	bLeftProcessed := FALSE;
	bRightProcessed := FALSE;
	bTransportBusy := FALSE;
	bUseDualGrip := FALSE;
	UseBoxCamera := FALSE;
	bLeftPlateArrived := FALSE;
	bRightPlateArrived := FALSE;
	bLeftPlateDone := FALSE;
	bRightPlateDone := FALSE;
	bLeftPlateReady_Prev := FALSE;
	bRightPlateReady_Prev := FALSE;
	bLeftConfigLatched := FALSE;
	bRightConfigLatched := FALSE;
	bLeftConfigReady_Prev := FALSE;
	bRightConfigReady_Prev := FALSE;

	uiExecutingStep := 50;
50:
	Cylinder.List.fbSameSizeCV_Press3.M_Extend();
	Cylinder.List.fbSameSizeCV_Press1.M_Extend();
	IF 	Cylinder.List.fbSameSizeCV_Press3.InFrontPosition
		AND	Cylinder.List.fbSameSizeCV_Press1.infrontposition
	THEN
		uiExecutingStep := 100;
	END_IF
// ═══════════════════════════════════════════════════
// Step 100: 三軌平行運行
// ═══════════════════════════════════════════════════
100:
	// C# 信號已透過 VAR_INPUT 傳入，不需要 HandShake reference 檢查

	// ================================================================
	// Track 1: 小手臂取盒 (鐵盤 → 同尺寸軌道)
	// ================================================================
	CASE uiPickStep OF
		0:	// 初始化
			bLeftProcessed 		:= FALSE;
			bRightProcessed 	:= FALSE;
			bPickTrackDone 		:= FALSE;
			bLeftPlateDone 		:= FALSE;
			bRightPlateDone 	:= FALSE;
			bLeftPlateArrived 	:= FALSE;
			bRightPlateArrived 	:= FALSE;
			uiPickStep := 100;

		100:	// 等待鐵盤到位
			// 偵測到位 (上升沿) — 目前由 C# ADS 模擬寫入, 後續要改成獨立硬體訊號
			IF bLeftPlateReady AND NOT bLeftPlateReady_Prev THEN
				bLeftPlateArrived := TRUE;
				bLeftProcessed := FALSE;
				bLeftPlateDone := FALSE;		// [Fix H2] 新盤到位，清除上一盤 Done
			END_IF
			IF bRightPlateReady AND NOT bRightPlateReady_Prev THEN
				bRightPlateArrived := TRUE;
				bRightProcessed := FALSE;
				bRightPlateDone := FALSE;		// [Fix H2]
			END_IF
			bLeftPlateReady_Prev := bLeftPlateReady;
			bRightPlateReady_Prev := bRightPlateReady;

			// [Fix H1] ConfigReady 上升沿鎖存
			IF bLeftConfigReady AND NOT bLeftConfigReady_Prev THEN
				bLeftConfigLatched := TRUE;
			END_IF
			IF bRightConfigReady AND NOT bRightConfigReady_Prev THEN
				bRightConfigLatched := TRUE;
			END_IF
			bLeftConfigReady_Prev := bLeftConfigReady;
			bRightConfigReady_Prev := bRightConfigReady;

			// 兩邊都 OFF → Done 計時
			TON_PlateWaitTimeout.IN := NOT bLeftPlateReady AND NOT bRightPlateReady
										AND NOT bLeftPlateArrived AND NOT bRightPlateArrived;

			// 有盤到位且 C# 已給配置 → 開始取盒 (先左後右)
			IF bLeftPlateReady AND bLeftConfigLatched AND NOT bLeftProcessed THEN
				bLeftPlateArrived := FALSE;
				bLeftConfigLatched := FALSE;
				uiCurrentSide := 0;
				uiCurrentSlot := 0;
				TON_ConfigTimeout.IN := FALSE;
				uiPickStep := 200;
			ELSIF bRightPlateReady AND bRightConfigLatched AND NOT bRightProcessed THEN
				bRightPlateArrived := FALSE;
				bRightConfigLatched := FALSE;
				uiCurrentSide := 1;
				uiCurrentSlot := 0;
				TON_ConfigTimeout.IN := FALSE;
				uiPickStep := 200;
			END_IF

			// 等待 C# 配置逾時
			IF (bLeftPlateArrived OR bRightPlateArrived) THEN
				TON_ConfigTimeout.IN := TRUE;
				IF TON_ConfigTimeout.Q THEN
					uiResumePickStep := uiPickStep;
					uiResumeCameraStep := uiCameraStep;
					uiResumeTransportStep := uiTransportStep;
					strStatus := 'FB_SameSizeCV_ReverseBatchPickAndPhoto Step 100: Waiting C# plate config timeout';
					_UniqueErrorCode := 'E_CONFIG_TIMEOUT';
					_Abort := TRUE;
					RETURN;
				END_IF
			END_IF

		200:	// 尋找下一個要取的格子
			IF uiCurrentSide = 0 THEN
				WHILE uiCurrentSlot <= 3 AND NOT LeftPlate[uiCurrentSlot] DO
					uiCurrentSlot := uiCurrentSlot + 1;
				END_WHILE
			ELSE
				WHILE uiCurrentSlot <= 3 AND NOT RightPlate[uiCurrentSlot] DO
					uiCurrentSlot := uiCurrentSlot + 1;
				END_WHILE
			END_IF

			IF uiCurrentSlot > 3 THEN
				uiPickStep := 500;
			ELSIF uiUnphotographedCount < 5 THEN
				uiPickStep := 300;
			ELSE
				uiPickStep := 250;
			END_IF

		250:	// 等待軌道空間
			IF uiUnphotographedCount < 5 THEN
				uiPickStep := 300;
			END_IF

		300:	// 啟動小手臂
			ShippingTransfer.Info.Source.Area := SEL(uiCurrentSide = 0,
			E_RobotArea.ShippingRobotRight, E_RobotArea.ShippingRobotLeft);
			ShippingTransfer.Info.Source.Position := UINT_TO_INT(uiCurrentSlot + 1);
			ShippingTransfer.Info.Source.Get := TRUE;
			ShippingTransfer.Info.Destination.Area := E_RobotArea.TransmitCV_End;
			ShippingTransfer.Info.Destination.Position := 1;
			ShippingTransfer.Info.Destination.Get := FALSE;
			uiPickStep := 305;
			
		305:
			ShippingTransfer.Execute := TRUE;
			uiPickStep := 310;

		310:	// 等待完成
			TON_PickupTimeout.IN := TRUE;
			IF ShippingTransfer.Done THEN
				TON_PickupTimeout.IN := FALSE;
				ShippingTransfer.Execute := FALSE;
				uiPickStep := 320;
			END_IF
			IF ShippingTransfer.Error OR ShippingTransfer.Aborted THEN
				TON_PickupTimeout.IN := FALSE;
				ShippingTransfer.Execute := FALSE;
				uiResumePickStep := 300;
				uiResumeCameraStep := uiCameraStep;
				uiResumeTransportStep := uiTransportStep;
				strStatus := 'FB_SameSizeCV_ReverseBatchPickAndPhoto Step 100: ShippingRobot pickup failed';
				_UniqueErrorCode := 'E_PICKUP_TIMEOUT';
				_Abort := TRUE;
				RETURN;
			END_IF
			IF TON_PickupTimeout.Q THEN
				ShippingTransfer.Execute := FALSE;
				uiResumePickStep := 300;
				uiResumeCameraStep := uiCameraStep;
				uiResumeTransportStep := uiTransportStep;
				strStatus := 'FB_SameSizeCV_ReverseBatchPickAndPhoto Step 100: ShippingRobot pickup timeout';
				_UniqueErrorCode := 'E_PICKUP_TIMEOUT';
				_Abort := TRUE;
				RETURN;
			END_IF

		320:	// 等待 DORMANT
			IF NOT ShippingTransfer.Busy AND NOT ShippingTransfer.Done THEN
				uiPickStep := 400;
			END_IF

		400:	// 更新計數，觸發拍照
			uiUnphotographedCount := uiUnphotographedCount + 1;
			uiTotalProcessed := uiTotalProcessed + 1;
			uiCameraRequestCount := uiCameraRequestCount + 1;
			uiCurrentSlot := uiCurrentSlot + 1;
			uiPickStep := 200;

		500:	// 本盤取完，通知 C#
			IF uiCurrentSide = 0 THEN
				bLeftPlateDone := TRUE;
				bLeftProcessed := TRUE;
			ELSE
				bRightPlateDone := TRUE;
				bRightProcessed := TRUE;
			END_IF

			// 檢查是否需要取另一盤
			IF uiCurrentSide = 0 AND bRightPlateReady AND bRightConfigLatched AND NOT bRightProcessed THEN
				bRightPlateArrived := FALSE;
				bRightConfigLatched := FALSE;
				uiCurrentSide := 1;
				uiCurrentSlot := 0;
				uiPickStep := 200;
			ELSE
				bPickTrackDone := TRUE;
				uiPickStep := 100;
			END_IF

	END_CASE

	// ================================================================
	// Track 2: 逆向拍照 (單盒 Handshake)
	// ================================================================
	CASE uiCameraStep OF
		0:	// 等待觸發
			IF uiCameraRequestCount > 0 THEN
				uiCameraRequestCount := uiCameraRequestCount - 1;
				uiCameraStep := 50;
			END_IF
		50:
			_fbSameSizeCV_ReverseCamera.xExecute := TRUE;
			UseBoxCamera := _fbSameSizeCV_ReverseCamera.UseBoxCamera;
			IF UseBoxCamera THEN
				uiCameraStep := 100;
			END_IF

		100:	// 等待 C# 拍照完成
			TON_CameraTimeout.IN := TRUE;
			IF BoxCameraDone THEN
				_fbSameSizeCV_ReverseCamera.BoxCameraDone := TRUE;
				TON_CameraTimeout.IN := FALSE;
				uiCameraStep := 150;
			END_IF
			IF TON_CameraTimeout.Q THEN
				uiResumePickStep := uiPickStep;
				uiResumeCameraStep := uiCameraStep;
				uiResumeTransportStep := uiTransportStep;
				strStatus := 'FB_SameSizeCV_ReverseBatchPickAndPhoto Step 100: Camera timeout';
				_UniqueErrorCode := 'E_CAMERA_TIMEOUT';
				_Abort := TRUE;
				RETURN;
			END_IF
			
		150:
			IF _fbSameSizeCV_ReverseCamera.xDone THEN
				_fbSameSizeCV_ReverseCamera.xExecute := FALSE;
			END_IF
			IF  NOT _fbSameSizeCV_ReverseCamera.xExecute 
				AND NOT _fbSameSizeCV_ReverseCamera.xBusy
				AND NOT _fbSameSizeCV_ReverseCamera.xError 
			THEN
				uiCameraStep := 200;
			END_IF

		200:	// 記錄結果到佇列
			UseBoxCamera := FALSE;

			IF BoxQueue.Count < 16 THEN
				uiUnphotographedCount := uiUnphotographedCount - 1;

				BoxQueue.Boxes[BoxQueue.WriteIdx].bActive 		:= TRUE;
				BoxQueue.Boxes[BoxQueue.WriteIdx].bIsOK 		:= CameraIsOK;
				BoxQueue.Boxes[BoxQueue.WriteIdx].iWarehouse 	:= CameraWarehouse;
				BoxQueue.Boxes[BoxQueue.WriteIdx].iLevel 		:= CameraLevel;
				BoxQueue.Boxes[BoxQueue.WriteIdx].iTrack 		:= CameraTrack;

				BoxQueue.WriteIdx := (BoxQueue.WriteIdx + 1) MOD 16;
				BoxQueue.Count := BoxQueue.Count + 1;
				TON_CameraClearTimeout.IN := TRUE;
				uiCameraStep := 210;
			ELSE
				uiResumePickStep := uiPickStep;
				uiResumeCameraStep := uiCameraStep;
				uiResumeTransportStep := uiTransportStep;
				strStatus := 'FB_SameSizeCV_ReverseBatchPickAndPhoto Step 100: Conveyor full (queue overflow)';
				_UniqueErrorCode := 'E_CONVEYOR_FULL';
				_Abort := TRUE;
				RETURN;
			END_IF

		210:	// 等待 C# 清除 BoxCameraDone
			IF NOT BoxCameraDone THEN
				TON_CameraClearTimeout.IN := FALSE;
				uiCameraStep := 0;
			END_IF
			IF TON_CameraClearTimeout.Q THEN
				TON_CameraClearTimeout.IN := FALSE;
				uiResumePickStep := uiPickStep;
				uiResumeCameraStep := uiCameraStep;
				uiResumeTransportStep := uiTransportStep;
				strStatus := 'FB_SameSizeCV_ReverseBatchPickAndPhoto Step 100: C# did not clear BoxCameraDone';
				_UniqueErrorCode := 'E_CAMERA_CLEAR_TIMEOUT';
				_Abort := TRUE;
				RETURN;
			END_IF

	END_CASE

	// ================================================================
	// Track 3: 大手臂搬運 (透過 FB_SameSizeCV_ReverseBoxToWareHouse)
	// ================================================================
	CASE uiTransportStep OF
		0:	// 等待佇列有盒子
			IF BoxQueue.Count >= 2 THEN
				TON_WaitPairTimeout.IN := FALSE;
				bUseDualGrip := TRUE;
				uiTransportStep := 100;
			ELSIF BoxQueue.Count = 1 THEN
				TON_WaitPairTimeout.IN := TRUE;
				IF TON_WaitPairTimeout.Q THEN
					TON_WaitPairTimeout.IN := FALSE;
					bUseDualGrip := FALSE;
					uiTransportStep := 100;
				END_IF
			ELSE
				TON_WaitPairTimeout.IN := FALSE;
			END_IF

		100:	// 從佇列取出盒子
			stGripA := BoxQueue.Boxes[BoxQueue.ReadIdx];
			BoxQueue.Boxes[BoxQueue.ReadIdx].bActive := FALSE;
			BoxQueue.ReadIdx := (BoxQueue.ReadIdx + 1) MOD 16;
			BoxQueue.Count := BoxQueue.Count - 1;

			IF bUseDualGrip AND BoxQueue.Count > 0 THEN
				stGripB := BoxQueue.Boxes[BoxQueue.ReadIdx];
				BoxQueue.Boxes[BoxQueue.ReadIdx].bActive := FALSE;
				BoxQueue.ReadIdx := (BoxQueue.ReadIdx + 1) MOD 16;
				BoxQueue.Count := BoxQueue.Count - 1;
			ELSE
				stGripB.bActive := FALSE;
				bUseDualGrip := FALSE;
			END_IF

			bTransportBusy := TRUE;
			uiTransportStep := 200;

		200:	// 啟動 BoxToWareHouse — Batch 拍照流程 bIsOK 二分:TRUE=WareHouse / FALSE=NGConveyor (不走 PullOut)
			BoxToWareHouse.bBoxA_Enable		:= TRUE;
			IF stGripA.bIsOK THEN
				BoxToWareHouse.eBoxA_Destination := E_ReverseBoxDestination.WareHouse;
			ELSE
				BoxToWareHouse.eBoxA_Destination := E_ReverseBoxDestination.NGConveyor;
			END_IF
			BoxToWareHouse.iBoxA_Warehouse	:= stGripA.iWarehouse;
			BoxToWareHouse.iBoxA_Level		:= stGripA.iLevel;
			BoxToWareHouse.iBoxA_Track		:= stGripA.iTrack;

			BoxToWareHouse.bBoxB_Enable		:= bUseDualGrip;
			IF bUseDualGrip THEN
				IF stGripB.bIsOK THEN
					BoxToWareHouse.eBoxB_Destination := E_ReverseBoxDestination.WareHouse;
				ELSE
					BoxToWareHouse.eBoxB_Destination := E_ReverseBoxDestination.NGConveyor;
				END_IF
				BoxToWareHouse.iBoxB_Warehouse	:= stGripB.iWarehouse;
				BoxToWareHouse.iBoxB_Level		:= stGripB.iLevel;
				BoxToWareHouse.iBoxB_Track		:= stGripB.iTrack;
			END_IF
			uiTransportStep := 205;
			
		205:

			BoxToWareHouse.Execute := TRUE;
			uiTransportStep := 300;

		300:	// 等待完成
			IF BoxToWareHouse.Done THEN
				BoxToWareHouse.Execute := FALSE;
				uiTransportedCount := uiTransportedCount + 1;
				IF bUseDualGrip THEN
					uiTransportedCount := uiTransportedCount + 1;
				END_IF
				uiTransportStep := 400;
			END_IF
			IF BoxToWareHouse.Error OR BoxToWareHouse.Aborted THEN
				BoxToWareHouse.Execute := FALSE;
				uiResumePickStep := uiPickStep;
				uiResumeCameraStep := uiCameraStep;
				uiResumeTransportStep := 200;
				strStatus := 'FB_SameSizeCV_ReverseBatchPickAndPhoto Step 100: BigArm transport failed';
				_UniqueErrorCode := 'E_BIGARM_TIMEOUT';
				_Abort := TRUE;
				RETURN;
			END_IF

		400:	// 等待子 FB 回到 DORMANT
			IF NOT BoxToWareHouse.Busy AND NOT BoxToWareHouse.Done THEN
				uiTransportStep := 500;
			END_IF

		500:	// 回到待命
			bTransportBusy := FALSE;
			stGripA.bActive := FALSE;
			stGripB.bActive := FALSE;
			uiTransportStep := 0;

	END_CASE

	// ================================================================
	// Done 判斷
	// ================================================================
	IF TON_PlateWaitTimeout.Q
	   AND uiUnphotographedCount = 0
	   AND BoxQueue.Count = 0
	   AND NOT bTransportBusy
	   AND uiTotalProcessed > 0
	   AND uiTotalProcessed = uiTransportedCount THEN
		_Executed := TRUE;
	END_IF

END_CASE

// 狀態切換
IF _Error THEN
	eState := STATE_ERROR;
ELSIF _Abort THEN
	eState := STATE_ABORTING;
ELSIF _Executed THEN
	eState := STATE_DONE;
ELSIF NOT Execute THEN
	estate := STATE_RESETTING;
END_IF
END_METHOD

// 重置狀態 — 清除旗標，支援 Retry/Resume
METHOD M_STATE_RESETTING
VAR_INPUT
END_VAR
Busy := TRUE;
Error := FALSE;
Aborted := FALSE;

CASE uiResettingStep OF
0:
	tonTimeOut.IN := FALSE;

	// 清除所有 Timer
	TON_PlateWaitTimeout.IN		:= FALSE;
	TON_PickupTimeout.IN		:= FALSE;
	TON_CameraTimeout.IN		:= FALSE;
	TON_ConfigTimeout.IN		:= FALSE;
	TON_WaitPairTimeout.IN		:= FALSE;
	TON_CameraClearTimeout.IN	:= FALSE;

	Cylinder.List.fbSameSizeCV_Press3.M_Retract();
	Cylinder.List.fbSameSizeCV_Press1.M_Retract();

	_fbSameSizeCV_ReverseCamera.xExecute := FALSE;
//	// _bRetry: 從 ABORTED 觸發 → 恢復到中斷點繼續
//	IF _bRetry THEN
//		_bRetry := FALSE;

//		eState := STATE_EXECUTING;
//		RETURN;
//	END_IF

	uiResettingStep := 100;

100:
	Done := FALSE;
	Busy := FALSE;
	_ResetCompleted := TRUE;
END_CASE

IF _ResetCompleted AND NOT Execute THEN
	eState := STATE_DORMANT;
END_IF
END_METHOD

END_FUNCTION_BLOCK

// ---- Library/20_MachineUnits/21_StorageArea/210_Cabinet/FB_WareHouse.TcPOU
FUNCTION_BLOCK FB_WareHouse EXTENDS FB_Objectbase
VAR_INPUT
	 Motors 		  : REFERENCE TO UNI_MotorList;
	 WheelhouseSensor : REFERENCE TO UNI_HMI_WheelHouseInput;
END_VAR
VAR_OUTPUT
END_VAR
VAR
   
    nMotorIndex    : UINT;
    CabinetJob     : E_CabinetJob := E_CabinetJob.Idle;    

    stLayerStatus    : st_LayerStatus;
    stWarehouseLayer : st_WarehouseLayer;
    stWarehouseList  : st_WarehouseList;
    _stWarehouseList : _st_WarehouseList;

	fbReloadBox : FB_ReloadBox;
	fbFeedInBox : FB_FeedInBox;
END_VAR

SUPER^.M_clcUpdate();
THIS^.M_clcUpdate();

PROPERTY PUBLIC bFeedInBox_Completed : BOOL
GET
bFeedInBox_Completed := fbFeedInBox.Done;
END_GET
END_PROPERTY

PROPERTY bReloadBox_Completed : BOOL
GET
bReloadBox_Completed := fbReloadBox.Done;
END_GET
END_PROPERTY

METHOD M_clcFBs : BOOL
VAR_INPUT	
END_VAR
VAR
	nELIndex			:	INT;
END_VAR
fbReloadBox(
	Execute:= , 
	Abort:= , 
	Reset:= , 
	ObjectName:= 'Warehouse Reload box', 
	Busy=> bBusy, 
	Done=> bDone, 
	Aborted=> , 
	Error=> bError, 
	ErrorID=> , 
	Status=> , 
	Motors:= Motors,
	WarehouseStatus:= WheelhouseSensor.List,
	ArrivedDelayTime:= T#1S,
	WarehouseSelect:= ,
	WarehouseCoordinates:= ,
	TimeOut:= T#10S);

fbFeedInBox(
	Execute:= ,
	Abort:= ,
	Reset:= ,
	ObjectName:= 'Warehouse FeedIn box',
	Busy=> bBusy,
	Done=> bDone,
	Aborted=> ,
	Error=> bError,
	ErrorID=> ,
	Status=> ,
	Motors:= Motors,
	WarehouseStatus:= WheelhouseSensor.List,
	ArrivedDelayTime:= T#2S,
	WarehouseSelect:= ,
	WarehouseCoordinates:= ,
	TimeOut:= T#10S);
END_METHOD

METHOD M_clcUpdate : BOOL
VAR_INPUT	
END_VAR
VAR	
	i : INT;
END_VAR
//clc FBs
M_clcFBs();
END_METHOD

METHOD PRIVATE M_GotoCommandStep : BOOL
VAR_INPUT
END_VAR
CabinetJob := E_CabinetJob.Initial;
END_METHOD

METHOD PRIVATE M_GotoErrorStep : BOOL
VAR_INPUT
END_VAR
CabinetJob := E_CabinetJob.error;
END_METHOD

METHOD PUBLIC M_ResetFeedInBox : BOOL
VAR_INPUT
END_VAR
VAR
	uiMotorInder : UINT; 
END_VAR
// reset reload box execute
fbFeedInBox.Execute := FALSE;
 
M_ResetFeedInBox := TRUE; // Method end
END_METHOD

METHOD M_ResetReloadBox : Bool
VAR_INPUT
END_VAR
// reset reload box execute
fbReloadBox.Execute := FALSE;

M_ResetReloadBox := true; // Method end
END_METHOD

METHOD PUBLIC M_StartFeedInBox : BOOL
VAR_INPUT
	WareHouseSelect : E_WareHouse;
	WarehouseCoordinates : ST_WareHouseCoordinates;
END_VAR
// Send command to Feedin box fb
fbFeedInBox.WarehouseSelect := WareHouseSelect;
fbFeedInBox.WarehouseCoordinates := WarehouseCoordinates;
fbFeedInBox.Execute := TRUE;

M_StartFeedInBox := TRUE; // Method end
END_METHOD

METHOD M_StartReloadBox : BOOL
VAR_INPUT
	WareHouseSelect : E_WareHouse;
	WarehouseCoordinates : ST_WareHouseCoordinates;
END_VAR
// Send command to reload box fb
fbReloadBox.WarehouseSelect := WareHouseSelect;
fbReloadBox.WarehouseCoordinates := WarehouseCoordinates;
fbReloadBox.Execute := TRUE;

M_StartReloadBox := true; // Method end
END_METHOD

END_FUNCTION_BLOCK

// ---- Library/20_MachineUnits/21_StorageArea/210_Cabinet/Services/FB_ReloadBox.TcPOU
FUNCTION_BLOCK FB_ReloadBox EXTENDS FB_ObjectBase_V2 IMPLEMENTS IBasicElement
VAR_INPUT
	Motors : REFERENCE TO UNI_MotorList ;// The motors with warehouse conveyor
	WarehouseStatus : REFERENCE TO ST_WheelhouseInput; // The warehouse motor and sensor status
	ArrivedDelayTime : TIME;
	WarehouseSelect :E_WareHouse;
	WarehouseCoordinates : ST_WareHouseCoordinates;
	TimeOut : TIME; // Set the time if the process stop
END_VAR
VAR_OUTPUT
END_VAR
VAR
	Ton_ArriveDelay : TON; // When box arrived the front sensor, delay some time.
	Ton_BoxMoveForward : TON;// When the conveyor send the box forward, but not useful.
	uiMotorIndex: INT;
	CurrentTargetSensorStatus : BOOL;
END_VAR

A00_BasicUnits();
A10_StateControl();

ACTION A00_BasicUnits:
// Timer
Ton_ArriveDelay(PT:= ArrivedDelayTime);
Ton_BoxMoveForward(PT:= TimeOut);
END_ACTION

(* Check Warehouse front sensor status
*)
METHOD M_CheckSlideSensor
VAR_INPUT
    WarehouseSelect      : E_WareHouse;
    WarehouseCoordinates : ST_WareHouseCoordinates;
END_VAR
VAR_OUTPUT
	SensorStatus : BOOL;
END_VAR
IF WarehouseSelect = E_WareHouse.WareHouseA THEN
    SensorStatus := WarehouseStatus.WheelhouseA.arLayer[WarehouseCoordinates.Layer].Line[WarehouseCoordinates.Slide];
ELSIF WarehouseSelect = E_WareHouse.WareHouseB THEN
    SensorStatus := WarehouseStatus.WheelhouseB.arLayer[WarehouseCoordinates.Layer].Line[WarehouseCoordinates.Slide];
END_IF
END_METHOD

METHOD  M_STATE_ABORTED
VAR_INPUT
END_VAR
END_METHOD

METHOD  M_STATE_ABORTING
VAR_INPUT
END_VAR
END_METHOD

METHOD  M_STATE_DONE
VAR_INPUT
END_VAR
Busy := FALSE;
Done := _Executed;
IF NOT Execute THEN
	eState := STATE_RESETTING;
END_IF
END_METHOD

METHOD  M_STATE_DORMANT
VAR_INPUT
END_VAR
// Clear FB output
Busy            := FALSE;
Done            := FALSE;
Aborted         := FALSE;
Error           := FALSE;
ErrorID         := 0;
Status          := '';
_ResetCompleted := FALSE;
_Error          := FALSE;
_Executed       := FALSE;
Ton_ArriveDelay.IN := FALSE;
Ton_BoxMoveForward.IN := FALSE;
uiExecutingStep := 0;
CurrentTargetSensorStatus := FALSE;
// Wait Execute command
IF Execute THEN
    eState := STATE_EXECUTING;
END_IF
END_METHOD

METHOD  M_STATE_ERROR
VAR_INPUT
END_VAR
FOR uiMotorIndex := 1 TO 20 DO
	Motors.arMotor[uiMotorIndex].M_MotorStop();// 
END_FOR

IF NOT Execute THEN
	estate := STATE_RESETTING;
END_IF
END_METHOD

METHOD  M_STATE_EXECUTING
VAR_INPUT
END_VAR
VAR_INST
	TargetLayer : INT;
	TargetSlide :E_WareHouseSlide;
END_VAR
// Set FB state is busy
Busy := TRUE;

// Process
CASE uiExecutingStep OF
    0: // Command analize
		 Ton_ArriveDelay.IN := FALSE;
		 TargetLayer := WarehouseCoordinates.Layer+(WarehouseSelect-1)*10; //Warehouse A = 1 , B = 2
		 TargetSlide := WarehouseCoordinates.Slide;
		uiExecutingStep := 10;
	10:
		 Ton_BoxMoveForward.IN := TRUE;
        Motors.arMotor[TargetLayer].M_MoveForward();// .M_MoveForward();//('Reload box : conveyor move forward');
		IF NOT Motors.arMotor[TargetLayer].InStopped THEN// .InStopped;// THEN
			Ton_BoxMoveForward.IN := FALSE;
			uiExecutingStep := 100;
		END_IF
		IF  Ton_BoxMoveForward.Q THEN
		  _Error := TRUE;
           Status := 'FB_ReloadBox Step 10: Move motor timeout';
		END_IF
    100: // Wait box arrived
        Ton_BoxMoveForward.IN := TRUE;
		M_CheckSlideSensor(WarehouseSelect := WarehouseSelect, WarehouseCoordinates := WarehouseCoordinates,SensorStatus=>CurrentTargetSensorStatus);
        Ton_ArriveDelay.IN:=CurrentTargetSensorStatus;

		IF Ton_ArriveDelay.Q THEN
            uiExecutingStep := 200;
//        ELSIF Ton_BoxMoveForward.Q THEN
//            _Error := TRUE;
//            Status := 'Box was not been arrived,time out';
        END_IF
    200:
        Ton_ArriveDelay.IN := FALSE;

        //IF Ton_ArriveDelay.Q THEN
            uiExecutingStep := 300;
       // END_IF
    300:
        Motors.arMotor[TargetLayer].M_MotorStop();// .M_MotorStop();//('Reload box : conveyor move forward');
        uiExecutingStep := 9900;
    9900:
        // Command completed
        _Executed := TRUE;
END_CASE

IF _Executed THEN
    eState := STATE_DONE;
ELSIF NOT Execute THEN
    eState := STATE_RESETTING;
ELSIF _Error THEN
    eState := STATE_ERROR;
END_IF
END_METHOD

METHOD  M_STATE_RESETTING
VAR_INPUT
END_VAR
VAR 
	uiMotorIndex : UINT;
END_VAR
Done := _Executed;
		Ton_BoxMoveForward.IN := FALSE;
		Ton_ArriveDelay.IN := FALSE;
FOR uiMotorIndex := 1 TO 20 DO 
	Motors.arMotor[uiMotorIndex].M_MotorStop();
END_FOR		
		
IF NOT Execute THEN
	eState := STATE_DORMANT;
END_IF
END_METHOD

END_FUNCTION_BLOCK

// ---- Library/20_MachineUnits/21_StorageArea/210_Cabinet/Services/FB_FeedInBox.TcPOU
FUNCTION_BLOCK FB_FeedInBox EXTENDS FB_ObjectBase_V2 IMPLEMENTS IBasicElement
VAR_INPUT
	Motors : REFERENCE TO UNI_MotorList ; // The motors with warehouse conveyor
	WarehouseStatus : REFERENCE TO ST_WheelhouseInput; // The warehouse motor and sensor status
	ArrivedDelayTime : TIME;
	WarehouseSelect :E_WareHouse;
	WarehouseCoordinates : ST_WareHouseCoordinates;
	TimeOut : TIME; // Set the time if the process stop
END_VAR
VAR_OUTPUT
END_VAR
VAR
	Ton_ArriveDelay : TON; // When box arrived the front sensor, delay some time.
	Ton_BoxMoveForward : TON;// When the conveyor send the box forward, but not useful.
	tonFirstReserveTime	:TON;
	tonSecondForwardTime	:TON;
	tonThirdReserceTime	:TON;
	uiMotorIndex: INT;
	CurrentTargetSensorStatus : BOOL;
END_VAR

A00_BasicUnits();
A10_StateControl();

ACTION A00_BasicUnits:
// Timer
Ton_ArriveDelay(PT:= ArrivedDelayTime);//2.0s
Ton_BoxMoveForward(PT:= TimeOut);//10S

//check full box in cabinet time
tonFirstReserveTime(PT :=T#1.5S);
tonSecondForwardTime(PT :=T#750MS);
tonThirdReserceTime(PT := ArrivedDelayTime);
END_ACTION

(* Check Warehouse front sensor status
*)
METHOD M_CheckSlideSensor
VAR_INPUT
    WarehouseSelect      : E_WareHouse;
    WarehouseCoordinates : ST_WareHouseCoordinates;
END_VAR
VAR_OUTPUT
	SensorStatus : BOOL;
END_VAR
IF WarehouseSelect = E_WareHouse.WareHouseA THEN
    SensorStatus := WarehouseStatus.WheelhouseA.arLayer[WarehouseCoordinates.Layer].Line[WarehouseCoordinates.Slide];
ELSIF WarehouseSelect = E_WareHouse.WareHouseB THEN
    SensorStatus := WarehouseStatus.WheelhouseB.arLayer[WarehouseCoordinates.Layer].Line[WarehouseCoordinates.Slide];
END_IF
END_METHOD

METHOD  M_STATE_ABORTED
VAR_INPUT
END_VAR
END_METHOD

METHOD  M_STATE_ABORTING
VAR_INPUT
END_VAR
END_METHOD

METHOD  M_STATE_DONE
VAR_INPUT
END_VAR
Busy := FALSE;
Done := TRUE;
IF NOT Execute THEN
	eState := STATE_RESETTING;
END_IF
END_METHOD

METHOD  M_STATE_DORMANT
VAR_INPUT
END_VAR
// Clear FB output
Busy            := FALSE;
Done            := FALSE;
Aborted         := FALSE;
Error           := FALSE;
ErrorID         := 0;
Status          := '';
_ResetCompleted := FALSE;
_Error          := FALSE;
_Executed       := FALSE;
Ton_ArriveDelay.IN := FALSE;
Ton_BoxMoveForward.IN := FALSE;
tonFirstReserveTime.IN :=FALSE;
tonSecondForwardTime.IN :=FALSE;
tonThirdReserceTime.IN :=FALSE;
uiExecutingStep := 0;
CurrentTargetSensorStatus := FALSE;
// Wait Execute command
IF Execute THEN
    eState := STATE_EXECUTING;
END_IF
END_METHOD

METHOD  M_STATE_ERROR
VAR_INPUT
END_VAR
FOR uiMotorIndex := 1 TO 20 DO
	Motors.arMotor[uiMotorIndex].M_MotorStop();
END_FOR

IF NOT Execute THEN
	estate := STATE_RESETTING;
END_IF
END_METHOD

METHOD  M_STATE_EXECUTING
VAR_INPUT
END_VAR
VAR_INST
	TargetLayer : INT;
	TargetSlide :E_WareHouseSlide;
END_VAR
VAR
	them: INT;
END_VAR
// Set FB state is busy
Busy := TRUE;

// Process
CASE uiExecutingStep OF
    0: // Command analize
		Ton_BoxMoveForward.IN := FALSE;
		Ton_ArriveDelay.IN := FALSE;
		tonFirstReserveTime.IN :=FALSE;
		tonSecondForwardTime.IN :=FALSE;
		tonThirdReserceTime.IN :=FALSE;
		TargetLayer := WarehouseCoordinates.Layer+(WarehouseSelect-1)*10 ; // Warehouse A=1 , B = 2;
		TargetSlide := WarehouseCoordinates.Slide;
		//uiExecutingStep := 10;
		uiExecutingStep := 50;		//modify : just backward CV  edit 20251112 Min
		
	10:	//Motor reverse make sure have space can retreat
		Motors.arMotor[TargetLayer].M_MoveBackward();
		Ton_BoxMoveForward.IN := TRUE;
		IF NOT Motors.arMotor[TargetLayer].InStopped  THEN 
			uiExecutingStep := 15;
		END_IF
		IF Ton_BoxMoveForward.Q THEN
			_Error :=TRUE;
			Status :='FB_FeedInBox Step 10: Storage Cabinet MoveBackward motor timeout';
		END_IF
	15:	//Motor First reverse  then stop motor 
		tonFirstReserveTime.IN := TRUE;
		Ton_BoxMoveForward.IN := FALSE;
		IF tonFirstReserveTime.Q THEN
			tonFirstReserveTime.IN :=FALSE;
			Motors.arMotor[TargetLayer].M_MotorStop();// .M_MotorStop();//('FeedIn Motors.arMotor stop reverse');
			IF Motors.arMotor[TargetLayer].InStopped THEN
				uiExecutingStep := 20;
			END_IF
		END_IF
		
	20:	//Motor SecondForward check cabinet layer have't full box inside 
		Motors.arMotor[TargetLayer].M_MoveForward();// .M_MoveForward();//('FeedIn box : make sure have space can feedIn');
		Ton_BoxMoveForward.IN :=TRUE;
		IF NOT Motors.arMotor[TargetLayer].InStopped THEN
			uiExecutingStep := 25;
		END_IF
		IF Ton_BoxMoveForward.Q THEN
			_Error :=TRUE;
			Status :='FB_FeedInBox Step 20: Storage Cabinet MoveForward motor timeout';
		END_IF
		
	25:	//Motor second MoveForward  then stop motor
		tonSecondForwardTime.IN := TRUE;
		Ton_BoxMoveForward.IN := FALSE;
		IF tonSecondForwardTime.Q THEN
			tonSecondForwardTime.IN :=FALSE;
			Motors.arMotor[TargetLayer].M_MotorStop();//('');
			IF Motors.arMotor[TargetLayer].InStopped THEN
				uiExecutingStep :=30;
			END_IF
		END_IF
		
	30:	//check layer haven't full box behind
		M_CheckSlideSensor(WarehouseSelect := WarehouseSelect, 
						   WarehouseCoordinates := WarehouseCoordinates,
						   SensorStatus=>CurrentTargetSensorStatus);
		IF NOT  CurrentTargetSensorStatus THEN
			uiExecutingStep :=50;
		ELSE
			_Error :=TRUE;
			Status :='FB_FeedInBox Step 30: Storage Cabinet Layer full box inside ,plaease remove box ';
		END_IF	
		
	50:
        Motors.arMotor[TargetLayer].M_MoveBackward();// .M_MoveBackward();// ('FeedIn box : conveyor move backward');
		Ton_BoxMoveForward.IN := TRUE;
		IF  NOT Motors.arMotor[TargetLayer].InStopped THEN
			Ton_BoxMoveForward.IN := FALSE;	
			uiExecutingStep := 100;
		END_IF		
		IF  Ton_BoxMoveForward.Q THEN
		  _Error := TRUE;
           Status := 'FB_FeedInBox Step 50: Move motor timeout';
		END_IF
		
    100: // Wait box arrived
		M_CheckSlideSensor(WarehouseSelect := WarehouseSelect, 
						   WarehouseCoordinates := WarehouseCoordinates,
						   SensorStatus=>CurrentTargetSensorStatus);
        IF NOT CurrentTargetSensorStatus THEN
            uiExecutingStep := 200;
        END_IF
    200:// third reverse 
        tonThirdReserceTime.IN := TRUE;
        IF tonThirdReserceTime.Q THEN
			tonThirdReserceTime.IN :=FALSE;
            uiExecutingStep := 300;
        END_IF
    300:
        Motors.arMotor[TargetLayer].M_MotorStop();//('FeedIn box : conveyor stop move');
        uiExecutingStep := 9900;
    9900:
        // Command completed
        _Executed := TRUE;
END_CASE

IF _Executed THEN
    eState := STATE_DONE;
ELSIF NOT Execute THEN
    eState := STATE_RESETTING;
ELSIF _Error THEN
    eState := STATE_ERROR;
END_IF
END_METHOD

METHOD  M_STATE_RESETTING
VAR_INPUT
END_VAR
VAR 
	uiMotorIndex : UINT;
END_VAR
Done := _Executed;

FOR uiMotorIndex := 1 TO 20 DO 
	Motors.arMotor[uiMotorIndex].M_MotorStop();
END_FOR	
IF NOT Execute THEN
	eState := STATE_DORMANT;
END_IF
END_METHOD

END_FUNCTION_BLOCK

// ---- Library/20_MachineUnits/23_ShippingArea/RobotService/FB_ShippingRobotTransfer.TcPOU
FUNCTION_BLOCK FB_ShippingRobotTransfer EXTENDS FB_ObjectBase_V2
VAR_INPUT
	Robot		: REFERENCE TO FB_FanucRobot_Basic_V2;
	Info		: ST_ShippingRobotTransfer_Info;
	Stop		: BOOL;
	Input		: REFERENCE TO ST_InputTable;
	Output		: REFERENCE TO ST_OutputTable;
	Motor		: REFERENCE TO UNI_MotorList;
	SameSizeCVRequest : REFERENCE TO ST_SameSizeCVRequest;	// Phase 2 仲裁 (僅 SameSize / pos=1 用,DifferentSize 仍直接驅動)
	Cylinder	: REFERENCE TO UNI_CylinderList;
	Buzz		: REFERENCE TO BOOL;
	RedLamp		: REFERENCE TO BOOL;
	bCompleteRequest	: BOOL;
	fbShippingHomingBusy	: BOOL;
END_VAR
VAR_OUTPUT
	bTransCVInPosition_Left		: BOOL;
	bTransCVInPosition_Right	: BOOL;
END_VAR
VAR
	// Phase tracking
	_fromArea	: E_RobotArea;
	_fromPos	: INT;
	_fromGet	: BOOL;
	_toArea		: E_RobotArea;
	_toPos		: INT;
	_toGet		: BOOL;

	// Robot move
	BoxReady_1st	: BOOL;
	Address_A		: INT;
	Area			: E_RobotArea;

	// Timers
	TON_RobotActionTimeOut		: TON;
	TON_CheckRobotDoneTimeOut	: TON;
	TON_BlinkDelay				: TON;
	tonBoxArriveDelay			: TON;
	TON_MechTimeOut				: TON;	// 機構(氣缸/輸送帶/sensor)前置動作逾時 (30s)
	TON_ServiceWatchDog			: TON;	// 整個 Service 執行總時間看門狗 (3min)
	TON_RSR02HomingTimeOut		: TON;	// ABORTING Error 8 (Not in Home Pos) 走 RSR02 回 home 超時 (120s)

	// TransmitCVEnd
	SensorToBeCheck		: BIT;
	ConveyorMotor		: REFERENCE TO FB_Motor;
	bMoveConveyorForward	: BOOL;
	bMoveConveyorBackward	: BOOL;
	bIsSameSize			: BOOL;	// Phase 2:ConveyorMotor 指向 TransmitSameSideCV (Position=1) — A00 寫請求,而非直接驅動

	// Buffer cylinder
	uiGetStep	: UDINT;

	// Blink (Left/Right buzz)
	BuzzBlinker		: Blink;
	LightBlinker	: Blink;
	TrigBuzz		: R_TRIG;
	TrigLight		: R_TRIG;
	BlinkInfo		: ST_BlinkInfo;

	// Resume
	uiResumeStep	: UDINT;	// 與 uiExecutingStep 同型別，避免 step 98000 / 99000 等大數字溢位
	strStatus		: STRING;
	_UniqueErrorCode	: STRING;
	PreviousStrStatus	: STRING;
	PreviousErrorCode	: STRING;
	
	_bRetry			: BOOL;
	_bAbsMoveStarted	: BOOL;	// 真的呼叫過 M_StartRobotAbsMove 才置 TRUE，防 stale Done 造成 ghost completion
	uiAbortedStep		: UDINT;	// STATE_ABORTED 內 Error 8 RSR02 recovery sub-state counter

	// Error blinking 閃爍邏輯
	trigErrorReset		: R_TRIG;
	tonErrorResetDelay	: TON;
	bErrorBlinking		: BOOL;
	
	HasBufferArea		: BOOL := FALSE;		// 直接在這裡切換True/False 就能判斷程式內部是否有判斷緩衝區機構了。>> false 無機構，True 有機構
END_VAR

A00_BasicUnits();
SUPER^.A10_StateControl();

ACTION A00_BasicUnits:
TON_RobotActionTimeOut(PT := T#60S);
TON_CheckRobotDoneTimeOut(PT := T#30S);
TON_BlinkDelay(PT := T#1S);
tonBoxArriveDelay(PT := T#1S);
TON_MechTimeOut(PT := T#30S);
TON_ServiceWatchDog(PT := T#180S);	// 3 分鐘總 Service 看門狗
TON_RSR02HomingTimeOut(PT := T#120S);	// ABORTING Error 8 RSR02 回 home 超時

// TransCV InPosition sensor 回饋 (左/右分開)
IF GVL_HMI.Setup.ShippingRobot_DockTestSignal THEN
	bTransCVInPosition_Left  := TRUE;
	bTransCVInPosition_Right := TRUE;
ELSE
	bTransCVInPosition_Left  := Input.bShippingTransCV_Leftside_Arrived;
	bTransCVInPosition_Right := Input.bShippingTransCV_Rightside_Arrived;
END_IF

// 輸送帶持續驅動邏輯 (Phase 2)
// SameSize:Busy 期間寫請求,由 FB_MachineControl.A20_ConveyorArbitration 驅動;非 Busy 不寫,避免本 FB 兩個 instance 互相 stomp。
// DifferentSize:本地直接驅動。
IF bIsSameSize THEN
	IF Busy AND __ISVALIDREF(SameSizeCVRequest) THEN
		SameSizeCVRequest.bShippingTransfer_NeedForward  := bMoveConveyorForward;
		SameSizeCVRequest.bShippingTransfer_NeedBackward := bMoveConveyorBackward;
	END_IF
ELSE
	IF bMoveConveyorForward AND __ISVALIDREF(ConveyorMotor) THEN
		IF NOT ConveyorMotor.InBackWard THEN
			ConveyorMotor.M_MoveForward();
		END_IF
	END_IF
	IF bMoveConveyorBackward AND __ISVALIDREF(ConveyorMotor) THEN
		IF NOT ConveyorMotor.InForWard THEN
			ConveyorMotor.M_MoveBackward();
		END_IF
	END_IF
END_IF
END_ACTION

METHOD M_CheckMechanism : BOOL
VAR_INPUT
END_VAR
IF HasBufferArea THEN
	M_CheckMechanism := TRUE;
	RETURN;
END_IF

IF (info.Destination.Area = E_RobotArea.ShippingBufferArea) OR
   (info.Source.Area = E_RobotArea.ShippingBufferArea) THEN
	M_CheckMechanism := FALSE;
	strStatus := 'FB_ShippingRobotTransfer: Wrong Command, no BufferArea';
	RETURN;
END_IF

M_CheckMechanism := TRUE;
END_METHOD

METHOD M_CheckTransferCommand : BOOL
VAR_INPUT
	AreaInfo : ST_ShippingRobotTransfer_AreaInfo;
END_VAR
M_CheckTransferCommand := FALSE;

CASE AreaInfo.Area OF
	E_RobotArea.ShippingRobotLeft,
	E_RobotArea.ShippingRobotRight:
		IF AreaInfo.Position < 1 OR AreaInfo.Position > 40 THEN
			strStatus := 'FB_ShippingRobotTransfer Step 100/7000: Wrong command, Left/Right Position must be 1-40';
			Status := strStatus;
			Error := TRUE;
			RETURN;
		END_IF

	E_RobotArea.ShippingBufferArea:
		IF AreaInfo.Position < 1 OR AreaInfo.Position > 55 THEN
			strStatus := 'FB_ShippingRobotTransfer Step 100/7000: Wrong command, Buffer Area Position must be 1-55';
			Status := strStatus;
			Error := TRUE;
			RETURN;
		END_IF

	E_RobotArea.TransmitCV_End:
		IF AreaInfo.Position < 1 OR AreaInfo.Position > 2 THEN
			strStatus := 'FB_ShippingRobotTransfer Step 100/7000: Wrong command, TransmitCV_End Position must be 1-2';
			Status := strStatus;
			Error := TRUE;
			RETURN;
		END_IF

	E_RobotArea.ShippingCCDPos:
		// CCD 位置固定 = 0，不需要檢查

	E_RobotArea.ShippingFeedOutEmptyBox:
		// 拔針排空盒位置固定 = 0
//		IF AreaInfo.Position <> 0 THEN
//			strStatus := 'FB_ShippingRobotTransfer Step 100/7000 : Wrong command, FeedOut Empty Box Position must be 0';
//			Status := strStatus;
//			Error := TRUE;
//			RETURN;
//		END_IF

ELSE
	strStatus := 'FB_ShippingRobotTransfer Step 100/7000: Wrong command, Invalid Area';
	Status := strStatus;
	Error := TRUE;
	RETURN;
END_CASE

 //檢查爪子狀態
IF AreaInfo.Get THEN
	// Get (取盒): 爪必須打開才能夾
	IF NOT Robot._DI1.ClampA_Open THEN
		strStatus := 'FB_ShippingRobotTransfer Step 100/7000: Wrong command, ClampA must be open to Get';
		Status := strStatus;
		Error := TRUE;
		RETURN;
	END_IF
ELSE
	// Put (放盒): 爪必須關閉 (夾著盒) 才能放
	IF Robot._DI1.ClampA_Open THEN
		strStatus := 'FB_ShippingRobotTransfer Step 100/7000: Wrong command, ClampA must be closed to Put';
		Status := strStatus;
		Error := TRUE;
		RETURN;
	END_IF
END_IF


M_CheckTransferCommand := TRUE;
END_METHOD

METHOD PRIVATE M_SensorUpdate
VAR_INPUT
	iPosition : INT;
END_VAR
CASE iPosition OF
1:
	SensorToBeCheck := Input.bSameSizeCV_BoxNearShippingSensor;
	ConveyorMotor REF= Motor.List.TransmitSameSideCV;
	bIsSameSize := TRUE;
2:
	SensorToBeCheck := Input.bDifferentSizeCV_BoxNearShippingSensor;
	ConveyorMotor REF= Motor.List.TransmitDifferentSideCV;
	bIsSameSize := FALSE;
END_CASE
END_METHOD

METHOD M_STATE_ABORTED
VAR_INPUT
END_VAR
IF NOT _bRetry THEN
	Busy  := FALSE;
	Error := TRUE;
	Aborted := TRUE;
	uiAbortingStep := 0;
	_AbortCompleted := FALSE;
END_IF

IF reset THEN
	_bRetry := TRUE;
	Error   := FALSE;
	Aborted := FALSE;
END_IF

IF NOT Execute THEN
	eState := STATE_RESETTING;
ELSIF Execute AND _bRetry THEN
	// Retry 兩分支:
	//   A. Robot 無 error  → 直接 resume EXECUTING (原本 retry 路徑)
	//   B. Robot 有 error  → 一律跑 RSR02 sub-state 回 home,完成後下個 cycle 走 A
	IF NOT Robot._DI1.Error THEN
		// 路徑 A
		uiExecutingStep := uiResumeStep;
		PreviousStrStatus := strStatus;
		PreviousErrorCode := _UniqueErrorCode;
		Status := 'FB_ShippingRobotTransfer: no error';
		_bRetry := FALSE;
		_bAbsMoveStarted := FALSE;
		uiAbortedStep := 0;
		eState := STATE_EXECUTING;
	ELSE
		// 路徑 B:任何 robot error 都走 RSR02 — 參考 FB_ShippingHoming step 500-1000 + FB_RobotSelfHoming step 302-318
		CASE uiAbortedStep OF
			0:	// 切 RSR02 命令手臂回 home
				Robot.OpMode := E_FanucRobotOpMode.RSR02;
				TON_RSR02HomingTimeOut.IN := TRUE;
				IF Robot._RSR2_Completed THEN
					TON_RSR02HomingTimeOut.IN := FALSE;
					uiAbortedStep := 100;
				ELSIF TON_RSR02HomingTimeOut.Q THEN
					// RSR02 超時:退回 ABORTED 等 user 介入
					TON_RSR02HomingTimeOut.IN := FALSE;
					strStatus := 'FB_ShippingRobotTransfer ABORTED: RSR02 homing timeout, manual intervention required';
					Status    := strStatus;
					_bRetry := FALSE;
					Error   := TRUE;
					Aborted := TRUE;
					uiAbortedStep := 0;
				END_IF
			100:	// 切回 RSR01 工作模式
				Robot.OpMode := E_FanucRobotOpMode.RSR01;
				IF Robot._RSR1_Ready THEN
					uiAbortedStep := 200;
				END_IF
			200:	// 確認 RSR01 切換完成 + 殘留 error 已清
				IF Robot.OpMode = E_FanucRobotOpMode.RSR01
					AND NOT Robot._DI1.Done
					AND Robot._DI12.RSR1_Active
					AND NOT Robot._DI1.Error
				THEN
					uiAbortedStep := 0;
					// 下一個 cycle 走路徑 A 自動 resume EXECUTING
				END_IF
		END_CASE
	END_IF
END_IF
END_METHOD

METHOD M_STATE_ABORTING
VAR_INPUT
END_VAR
CASE uiAbortingStep OF
	0:
			_Abort := FALSE;
			Abort  := FALSE;
			_bAbsMoveStarted := FALSE;	// Retry 前清掉 stale flag,避免 step 5000/15000 因 Done=TRUE 殘留誤判 ghost completion
			TON_RobotActionTimeOut.IN    := FALSE;
			TON_CheckRobotDoneTimeOut.IN := FALSE;
			TON_MechTimeOut.IN           := FALSE;
			TON_ServiceWatchDog.IN       := FALSE;
			TON_RSR02HomingTimeOut.IN    := FALSE;
			bMoveConveyorForward  := FALSE;
			bMoveConveyorBackward := FALSE;
			// Phase 2:SameSize 撤銷請求 (arbiter 自動停),DifferentSize 直接停
			IF bIsSameSize THEN
				IF __ISVALIDREF(SameSizeCVRequest) THEN
					SameSizeCVRequest.bShippingTransfer_NeedForward  := FALSE;
					SameSizeCVRequest.bShippingTransfer_NeedBackward := FALSE;
				END_IF
			ELSIF __ISVALIDREF(ConveyorMotor) THEN
				ConveyorMotor.M_MotorStop();
			END_IF
			// 中斷 robot AbsMove 命令，避免 abort 期間 robot 還在跑舊軌跡
			Robot.M_ResetRobotAbsMove(TRUE, FALSE);
			uiAbortingStep := 50;

	50:	// 等 robot 命令真的被 reset 掉再進入錯誤檢查
			TON_CheckRobotDoneTimeOut.IN := TRUE;
			IF NOT Robot._DI1.Done THEN
				TON_CheckRobotDoneTimeOut.IN := FALSE;
				uiAbortingStep := 100;
			ELSIF TON_CheckRobotDoneTimeOut.Q THEN
				// Reset 超時也繼續，後續 step 100 會處理 Robot.Error 路徑
				TON_CheckRobotDoneTimeOut.IN := FALSE;
				uiAbortingStep := 100;
			END_IF

	100:
			// 任何 robot error 都直接跳 9999 進 ABORTED;
			// 不在 ABORTING 嘗試一般 reset (200/300/400),所有 recovery 統一放在 ABORTED 內 user 按 reset 才執行 RSR02
			uiAbortingStep := 9999;

	9999:
		_AbortCompleted := TRUE;
END_CASE

IF _AbortCompleted THEN
	eState := STATE_ABORTED;
END_IF
END_METHOD

METHOD M_STATE_DONE
VAR_INPUT
END_VAR
Busy   := FALSE;
_Error := Error := FALSE;
_Abort := Abort := FALSE;
Done   := TRUE;

// Done 期間持續壓住所有輸出，防止任何旗標被 A00_BasicUnits 重新驅動
bMoveConveyorForward  := FALSE;
bMoveConveyorBackward := FALSE;
Buzz    := FALSE;
RedLamp := FALSE;

IF NOT Execute THEN
	eState := STATE_RESETTING;
END_IF
END_METHOD

METHOD M_STATE_DORMANT
VAR_INPUT
END_VAR
Busy            := FALSE;
Done            := FALSE;
Aborted         := FALSE;
Error           := FALSE;
Paused          := FALSE;
ErrorID         := 0;
Status          := '';
UniqueErrorCode := '';

_Executed            := FALSE;
_Error               := FALSE;
_Abort               := FALSE;
_ResetCompleted      := FALSE;
_AbortCompleted      := FALSE;
_HoldingCompleted    := FALSE;
_HeldCompleted       := FALSE;
_UnholdCompleted     := FALSE;
_bRetry              := FALSE;
_bAbsMoveStarted     := FALSE;

uiExecutingStep  := 0;
uiResettingStep  := 0;
uiAbortingStep   := 0;
uiHoldingStep    := 0;
uiHeldStep       := 0;
uiUnholdStep     := 0;
uiGetStep        := 0;
uiResumeStep     := 0;

TON_RobotActionTimeOut.IN    := FALSE;
TON_CheckRobotDoneTimeOut.IN := FALSE;
TON_BlinkDelay.IN            := FALSE;
tonBoxArriveDelay.IN         := FALSE;
TON_MechTimeOut.IN           := FALSE;
TON_ServiceWatchDog.IN       := FALSE;
TON_RSR02HomingTimeOut.IN    := FALSE;

bMoveConveyorForward  := FALSE;
bMoveConveyorBackward := FALSE;
bIsSameSize := FALSE;
// Phase 2:DORMANT 只清 local intent (bMoveConveyor*),不動 shared SameSizeCVRequest
// 本 FB 有兩個 instance,idle 不能 stomp 其他 instance 的 request。A00 已用 Busy gate 確保 idle 不寫 shared flag。
BoxReady_1st := FALSE;

// Buzz / Lamp 閃爍預設次數 (各 3 次 = 約 1.8 秒警示)
BlinkInfo.MaxBuzzCount  := 3;
BlinkInfo.MaxLightCount := 3;
BlinkInfo.BuzzCount     := 0;
BlinkInfo.LightCount    := 0;

Status := '';
Error := FALSE;
PreviousStrStatus := '';
PreviousErrorCode := '';
_UniqueErrorCode  := '0';

bCompleteRequest := FALSE;

IF Execute THEN
	IF M_CheckMechanism() THEN
		eState := STATE_EXECUTING;
	ELSE
		eState := STATE_ERROR;
	END_IF
END_IF
END_METHOD

METHOD M_STATE_ERROR
VAR_INPUT
END_VAR
// 預設錯誤/忙碌狀態輸出
Error  := TRUE;
Busy   := FALSE;
_Error := FALSE;
Status := strStatus;

// 停止各項輸出 (輸送帶等) — Phase 2 同 ABORTING
bMoveConveyorForward  := FALSE;
bMoveConveyorBackward := FALSE;
_bAbsMoveStarted := FALSE;	// 雙保險:ERROR 進入時清,避免下游若直接 retry 殘留 stale 旗標
IF bIsSameSize THEN
	IF __ISVALIDREF(SameSizeCVRequest) THEN
		SameSizeCVRequest.bShippingTransfer_NeedForward  := FALSE;
		SameSizeCVRequest.bShippingTransfer_NeedBackward := FALSE;
	END_IF
ELSIF __ISVALIDREF(ConveyorMotor) THEN
	ConveyorMotor.M_MotorStop();
END_IF

// --- Reset 閃爍邏輯：偵測上升緣觸發 1 秒閃爍 ---
trigErrorReset(CLK := reset);
IF trigErrorReset.Q THEN
	bErrorBlinking := TRUE;
END_IF

tonErrorResetDelay(IN := bErrorBlinking, PT := T#1S);
IF tonErrorResetDelay.Q THEN
	bErrorBlinking := FALSE;
END_IF

// 閃爍期間 (1秒) 暫時將 Error 訊號設為 FALSE
IF bErrorBlinking THEN
	Error := FALSE;
END_IF

// 只有當外部啟動訊號關閉時，才真正退出錯誤狀態並複歸
IF NOT Execute THEN
	Error := FALSE;
	bErrorBlinking := FALSE;
	tonErrorResetDelay.IN := FALSE;
	eState := STATE_RESETTING;
END_IF
END_METHOD

METHOD M_STATE_EXECUTING
VAR_INPUT
END_VAR
Busy := TRUE;

// 暫停
IF Pause THEN
	_HoldingCompleted  := FALSE;
	_HeldCompleted     := FALSE;
	_UnholdCompleted   := FALSE;
	uiHoldingStep      := 0;
	uiHeldStep         := 0;
	uiUnholdStep       := 0;
	eState := STATE_Holding;
	RETURN;
END_IF

// Service watchdog (3 分鐘總執行時間) — 持續跑到 99000 或 Abort / Stop
TON_ServiceWatchDog.IN := TRUE;

// Stop 時暫停 Timeout
IF THIS^.Stop THEN
	TON_RobotActionTimeOut.IN    := FALSE;
	TON_CheckRobotDoneTimeOut.IN := FALSE;
	TON_MechTimeOut.IN           := FALSE;
	TON_ServiceWatchDog.IN       := FALSE;
END_IF

// Service watchdog 逾時 → 整個 FB Abort + 報警
IF TON_ServiceWatchDog.Q THEN
	uiResumeStep := uiExecutingStep;
	strStatus    := 'FB_ShippingRobotTransfer: Service watchdog timeout (3 min)';
	Status       := strStatus;
	Error        := TRUE;
	_Abort       := TRUE;
END_IF

CASE uiExecutingStep OF

	// ============================================================
	// Phase 0: 初始化 + 命令驗證
	// ============================================================
	0:
		// 非自動模式直接報錯 (避免軸控衝突)
		IF GVL_Machine.PackTags[UnitNo.Shipping].Status.UnitModeCurrent <> E_UnitMode.Auto THEN
			strStatus := 'FB_ShippingRobotTransfer Step 0: Not in Auto mode';
			_UniqueErrorCode := 'E_NOT_AUTO_MODE';
			_Error := TRUE;
		ELSE
			// 清除變數
			BoxReady_1st          := FALSE;
			Address_A             := 0;
			uiGetStep             := 0;
			bMoveConveyorForward  := FALSE;
			bMoveConveyorBackward := FALSE;
			BlinkInfo.BuzzCount   := 0;
			BlinkInfo.LightCount  := 0;

			// 解析命令
			_fromArea := Info.Source.Area;
			_fromPos  := Info.Source.Position;
			_fromGet  := Info.Source.Get;
			_toArea   := Info.Destination.Area;
			_toPos    := Info.Destination.Position;
			_toGet    := Info.Destination.Get;
			
			uiExecutingStep := 25;
		END_IF

	25: // 指令邏輯驗證
		// 限制 1：來源 (Source) 必須是取件 (Get)，目的地 (Destination) 必須是放件 (Put)
		IF NOT _fromGet OR _toGet THEN
			strStatus := 'FB_ShippingRobotTransfer Step 25: Source must be "Get", Destination must be "Put"';
			_Error := TRUE;
		// 限制 2：ShippingFeedOutEmptyBox 不可作為來源 (Source)
		ELSIF _fromArea = E_RobotArea.ShippingFeedOutEmptyBox THEN
			strStatus := 'FB_ShippingRobotTransfer Step 25: ShippingFeedOutEmptyBox cannot be used as Source';
			_Error := TRUE;
		// 限制 3：目的地為 ShippingFeedOutEmptyBox 時，來源必須是 TransmitCV_End
		ELSIF _toArea = E_RobotArea.ShippingFeedOutEmptyBox AND _fromArea <> E_RobotArea.TransmitCV_End THEN
			strStatus := 'FB_ShippingRobotTransfer Step 25: ShippingFeedOutEmptyBox destination requires TransmitCV_End as source';
			_Error := TRUE;
		END_IF

		IF NOT _Error THEN
			uiExecutingStep := 50;
		END_IF

	50: // 檢查 TransCV InPosition (Source/Destination 若為 Left/Right 需對應旗標)
		// Source 檢查
		IF _fromArea = E_RobotArea.ShippingRobotLeft THEN
			IF NOT bTransCVInPosition_Left THEN
				uiResumeStep := 50;
				strStatus := 'FB_ShippingRobotTransfer Step 50: Source Left TransCV not in position';
				Status := strStatus;
				Error := TRUE;
				_Abort := TRUE;
			END_IF
		ELSIF _fromArea = E_RobotArea.ShippingRobotRight THEN
			IF NOT bTransCVInPosition_Right THEN
				uiResumeStep := 50;
				strStatus := 'FB_ShippingRobotTransfer Step 50: Source Right TransCV not in position';
				Status := strStatus;
				Error := TRUE;
				_Abort := TRUE;
			END_IF
		END_IF
		// Destination 檢查
		IF NOT _Abort THEN
			IF _toArea = E_RobotArea.ShippingRobotLeft THEN
				IF NOT bTransCVInPosition_Left THEN
					uiResumeStep := 50;
					strStatus := 'FB_ShippingRobotTransfer Step 50: Destination Left TransCV not in position';
					Status := strStatus;
					Error := TRUE;
					_Abort := TRUE;
				END_IF
			ELSIF _toArea = E_RobotArea.ShippingRobotRight THEN
				IF NOT bTransCVInPosition_Right THEN
					uiResumeStep := 50;
					strStatus := 'FB_ShippingRobotTransfer Step 50: Destination Right TransCV not in position';
					Status := strStatus;
					Error := TRUE;
					_Abort := TRUE;
				END_IF
			END_IF
		END_IF
		IF NOT _Abort THEN
			uiExecutingStep := 100;
		END_IF

	100: // 驗證 Source 命令
		IF M_CheckTransferCommand(Info.Source) THEN
			uiExecutingStep := 1000;
		ELSE
			_Error := TRUE;
		END_IF



	// ============================================================
	// Phase 1 (FROM): 區域前置作業
	// ============================================================
	1000: // FROM 區域分支
		Area      := _fromArea;
		Address_A := _fromPos;
		BoxReady_1st := FALSE;
		TON_RobotActionTimeOut.IN := FALSE;

		CASE _fromArea OF
			E_RobotArea.ShippingRobotLeft,
			E_RobotArea.ShippingRobotRight:
				// TransCV 已在 Step 50 檢查完畢
				uiExecutingStep := 5000;

			E_RobotArea.ShippingBufferArea:
				IF _fromGet THEN
					// Get from buffer - 位置55需氣缸
					uiExecutingStep := 1100;
				ELSE
					// Put to buffer - 確認氣缸縮回
					uiExecutingStep := 1200;
				END_IF

			E_RobotArea.TransmitCV_End:
				M_SensorUpdate(_fromPos);
				IF _fromGet THEN
					// Get: 啟動輸送帶正轉 (A00 propagates flag → arbiter/direct)
					bMoveConveyorForward := TRUE;
					uiExecutingStep := 5000;
				ELSE
					// Put: 啟動輸送帶反轉 + 等 sensor 清除
					bMoveConveyorBackward := TRUE;
					uiExecutingStep := 1300;
				END_IF

			E_RobotArea.ShippingCCDPos:
				// CCD 無前置作業
				Address_A := 0;
				uiExecutingStep := 5000;
		END_CASE

	1100: // Buffer Get 前置 - 氣缸處理
		TON_MechTimeOut.IN := TRUE;
		CASE uiGetStep OF
			0:
				CASE Address_A OF
					1..54:
						uiGetStep := 400;
					55:
						uiGetStep := 100;
				END_CASE
			100:
				Cylinder.List.fbShippingBuffer_Press.M_Extend();
				IF Cylinder.List.fbShippingBuffer_Press.InFrontPosition THEN
					uiGetStep := 300;
				END_IF
			300:
				Cylinder.List.fbShippingBuffer_Press.M_Retract();
				IF Cylinder.List.fbShippingBuffer_Press.InRearPosition THEN
					uiGetStep := 400;
				END_IF
			400:
				BoxReady_1st := TRUE;
				TON_MechTimeOut.IN := FALSE;
				uiExecutingStep := 5000;
		END_CASE
		IF TON_MechTimeOut.Q THEN
			uiResumeStep := 1100;
			strStatus := 'FB_ShippingRobotTransfer Step 1100: Buffer cylinder timeout';
			Status := strStatus;
			Error := TRUE;
			_Abort := TRUE;
		END_IF

	1200: // Buffer Put 前置 - 確認氣缸縮回
		TON_MechTimeOut.IN := TRUE;
		IF Cylinder.List.fbShippingBuffer_Press.InRearPosition THEN
			BoxReady_1st := TRUE;
			TON_MechTimeOut.IN := FALSE;
			uiExecutingStep := 5000;
		ELSE
			Cylinder.List.fbShippingBuffer_Press.M_Retract();
		END_IF
		IF TON_MechTimeOut.Q THEN
			uiResumeStep := 1200;
			strStatus := 'FB_ShippingRobotTransfer Step 1200: Buffer cylinder retract timeout';
			Status := strStatus;
			Error := TRUE;
			_Abort := TRUE;
		END_IF

	1300: // TransmitCVEnd Put 前置 - 等反轉 + sensor 清除
		TON_MechTimeOut.IN := TRUE;
		M_SensorUpdate(_fromPos);	// 每 scan 重新採樣 sensor，避免使用 step 1000 的舊值
		IF ConveyorMotor.InBackWard AND NOT SensorToBeCheck THEN
			TON_MechTimeOut.IN := FALSE;
			uiExecutingStep := 5000;
		END_IF
		IF TON_MechTimeOut.Q THEN
			uiResumeStep := 1300;
			strStatus := 'FB_ShippingRobotTransfer Step 1300: TransmitCV reverse / sensor clear timeout';
			Status := strStatus;
			Error := TRUE;
			_Abort := TRUE;
		END_IF

	// ============================================================
	// Phase 1 (FROM): Robot AbsMove + Reset
	// ============================================================
	5000: // Robot AbsMove
		TON_RobotActionTimeOut.IN := TRUE;
		IF NOT Robot._DI1.Done THEN
			// 正常路徑：robot 還在動 → 持續送 AbsMove 命令
			// TransmitCVEnd Get 時需要等 sensor
			IF Area = E_RobotArea.TransmitCV_End AND _fromGet THEN
				M_SensorUpdate(_fromPos);
				tonBoxArriveDelay.IN := SensorToBeCheck;
				bMoveConveyorForward := TRUE;
				Robot.M_StartRobotAbsMove(
					GetBox       := _fromGet,
					UseClampA    := TRUE,
					UseClampB    := FALSE,
					Area         := Area,
					ClampA_Address := Address_A,
					ClampB_Address := 0,
					BoxReady_1   := tonBoxArriveDelay.Q OR BoxReady_1st,
					BoxReady_2   := FALSE);
			ELSIF Area = E_RobotArea.ShippingCCDPos THEN
				// CCD 固定 GetBox=TRUE, Address=0
				Robot.M_StartRobotAbsMove(
					GetBox       := TRUE,
					UseClampA    := TRUE,
					UseClampB    := FALSE,
					Area         := Area,
					ClampA_Address := 0,
					ClampB_Address := 0,
					BoxReady_1   := BoxReady_1st,
					BoxReady_2   := FALSE);
			ELSE
				IF Area = E_RobotArea.ShippingBufferArea AND NOT _fromGet THEN
					// Buffer Put 已在前置設好 BoxReady
				ELSIF Area = E_RobotArea.ShippingBufferArea AND _fromGet THEN
					// Buffer Get 已在前置設好 BoxReady
				ELSE
					BoxReady_1st := TRUE;
				END_IF
				Robot.M_StartRobotAbsMove(
					GetBox       := _fromGet,
					UseClampA    := TRUE,
					UseClampB    := FALSE,
					Area         := Area,
					ClampA_Address := Address_A,
					ClampB_Address := 0,
					BoxReady_1   := BoxReady_1st,
					BoxReady_2   := FALSE);
			END_IF
			_bAbsMoveStarted := TRUE;	// 標記真的有送過 Start 命令
		ELSIF NOT _bAbsMoveStarted THEN
			// Done=TRUE 但從未送過 Start → stale 狀態（續做 / 上次殘留）
			// 先清掉 robot 命令，等 Done 變 FALSE 才能進入正常流程，避免 ghost completion
			Robot.M_ResetRobotAbsMove(TRUE, FALSE);
		ELSE
			// 真的完成（Done 從 FALSE → TRUE）→ 轉 5100
			// 不做手臂 ClampA_Sensor 驗證 — 軌道末端 BoxNearShippingSensor 已在 IF NOT Done 分支
			// 透過 tonBoxArriveDelay + BoxReady_1 把關取盒時機,robot 端確認結束後 PLC 直接信任 Done
			TON_RobotActionTimeOut.IN := FALSE;
			tonBoxArriveDelay.IN      := FALSE;
			_bAbsMoveStarted          := FALSE;
			uiExecutingStep := 5100;
		END_IF

		IF TON_RobotActionTimeOut.Q THEN
			uiResumeStep := 5000;
			strStatus := 'FB_ShippingRobotTransfer Step 5000: Robot AbsMove timeout';
			Status := strStatus;
			Error := TRUE;
			_Abort       := TRUE;
		END_IF
		IF Robot._DI1.Error THEN
			uiResumeStep := 5000;
			strStatus    := CONCAT('FROM: Robot Error ', Robot.ErrMsg);
			Status := strStatus;
			Error := TRUE;
			_Abort       := TRUE;
		END_IF

	5100: // FROM Reset Robot command
		Robot.M_ResetRobotAbsMove(TRUE, FALSE);
		TON_CheckRobotDoneTimeOut.IN := TRUE;
		IF NOT Robot._DI1.Done THEN
			TON_CheckRobotDoneTimeOut.IN := FALSE;
			uiExecutingStep := 6000;
		END_IF
		IF TON_CheckRobotDoneTimeOut.Q THEN
			uiResumeStep := 5100;
			strStatus := 'FB_ShippingRobotTransfer Step 5100: Robot Reset timeout';
			Status := strStatus;
			Error := TRUE;
			_Abort       := TRUE;
		END_IF
		IF Robot._DI1.Error THEN
			uiResumeStep := 5100;
			strStatus    := CONCAT('FROM Reset: Robot Error ', Robot.ErrMsg);
			Status := strStatus;
			Error := TRUE;
			_Abort       := TRUE;
		END_IF

	// ============================================================
	// Phase 1 (FROM): 區域後置作業
	// ============================================================
	6000: // FROM 後置
		// TransmitCVEnd: 停止輸送帶 — Phase 2 SameSize 撤銷請求,DifferentSize 直接停
		IF _fromArea = E_RobotArea.TransmitCV_End THEN
			bMoveConveyorForward  := FALSE;
			bMoveConveyorBackward := FALSE;
			IF bIsSameSize THEN
				IF __ISVALIDREF(SameSizeCVRequest) THEN
					SameSizeCVRequest.bShippingTransfer_NeedForward  := FALSE;
					SameSizeCVRequest.bShippingTransfer_NeedBackward := FALSE;
				END_IF
			ELSIF __ISVALIDREF(ConveyorMotor) THEN
				ConveyorMotor.M_MotorStop();
			END_IF
		END_IF

		// 重置變數準備 TO phase
		BoxReady_1st := FALSE;
		uiGetStep    := 0;
		_bAbsMoveStarted := FALSE;	// Phase 1 結束，重置 flag 給 Phase 2 step 15000 使用
		TON_RobotActionTimeOut.IN    := FALSE;
		TON_CheckRobotDoneTimeOut.IN := FALSE;
		uiExecutingStep := 7000;
		
	7000:
		IF M_CheckTransferCommand(Info.Destination) THEN
			uiExecutingStep := 10000;
		ELSE
			_Error := TRUE;
		END_IF

	// ============================================================
	// Phase 2 (TO): 區域前置作業
	// ============================================================
	10000: // TO 區域分支
		Area      := _toArea;
		Address_A := _toPos;
		BoxReady_1st := FALSE;

		CASE _toArea OF
			E_RobotArea.ShippingRobotLeft,
			E_RobotArea.ShippingRobotRight:
				// TransCV 已在 Step 50 檢查完畢
				uiExecutingStep := 15000;

			E_RobotArea.ShippingBufferArea:
				IF _toGet THEN
					uiExecutingStep := 10100;
				ELSE
					uiExecutingStep := 10200;
				END_IF

			E_RobotArea.TransmitCV_End:
				M_SensorUpdate(_toPos);
				IF _toGet THEN
					bMoveConveyorForward := TRUE;
					uiExecutingStep := 15000;
				ELSE
					bMoveConveyorBackward := TRUE;
					uiExecutingStep := 10300;
				END_IF

			E_RobotArea.ShippingCCDPos:
				Address_A := 0;
				uiExecutingStep := 15000;

			E_RobotArea.ShippingFeedOutEmptyBox:
				Address_A := _toPos;
				uiExecutingStep := 15000;
		END_CASE

	10100: // TO Buffer Get 前置
		TON_MechTimeOut.IN := TRUE;
		CASE uiGetStep OF
			0:
				CASE Address_A OF
					1..54:
						uiGetStep := 400;
					55:
						uiGetStep := 100;
				END_CASE
			100:
				Cylinder.List.fbShippingBuffer_Press.M_Extend();
				IF Cylinder.List.fbShippingBuffer_Press.InFrontPosition THEN
					uiGetStep := 300;
				END_IF
			300:
				Cylinder.List.fbShippingBuffer_Press.M_Retract();
				IF Cylinder.List.fbShippingBuffer_Press.InRearPosition THEN
					uiGetStep := 400;
				END_IF
			400:
				BoxReady_1st := TRUE;
				TON_MechTimeOut.IN := FALSE;
				uiExecutingStep := 15000;
		END_CASE
		IF TON_MechTimeOut.Q THEN
			uiResumeStep := 10100;
			strStatus := 'FB_ShippingRobotTransfer Step 10100: Buffer cylinder timeout';
			Status := strStatus;
			Error := TRUE;
			_Abort := TRUE;
		END_IF

	10200: // TO Buffer Put 前置
		TON_MechTimeOut.IN := TRUE;
		IF Cylinder.List.fbShippingBuffer_Press.InRearPosition THEN
			BoxReady_1st := TRUE;
			TON_MechTimeOut.IN := FALSE;
			uiExecutingStep := 15000;
		ELSE
			Cylinder.List.fbShippingBuffer_Press.M_Retract();
		END_IF
		IF TON_MechTimeOut.Q THEN
			uiResumeStep := 10200;
			strStatus := 'FB_ShippingRobotTransfer Step 10200: Buffer cylinder retract timeout';
			Status := strStatus;
			Error := TRUE;
			_Abort := TRUE;
		END_IF

	10300: // TO TransmitCVEnd Put 前置
		TON_MechTimeOut.IN := TRUE;
		M_SensorUpdate(_toPos);
		IF ConveyorMotor.InBackWard AND NOT SensorToBeCheck THEN
			TON_MechTimeOut.IN := FALSE;
			uiExecutingStep := 15000;
		END_IF
		IF TON_MechTimeOut.Q THEN
			uiResumeStep := 10300;
			strStatus := 'FB_ShippingRobotTransfer Step 10300: TransmitCV reverse / sensor clear timeout';
			Status := strStatus;
			Error := TRUE;
			_Abort := TRUE;
		END_IF

	// ============================================================
	// Phase 2 (TO): Robot AbsMove + Reset
	// ============================================================
	15000: // TO Robot AbsMove
		TON_RobotActionTimeOut.IN := TRUE;
		IF NOT Robot._DI1.Done THEN
			// 正常路徑：robot 還在動 → 持續送 AbsMove 命令
			IF Area = E_RobotArea.TransmitCV_End AND _toGet THEN
				M_SensorUpdate(_toPos);
				tonBoxArriveDelay.IN := SensorToBeCheck;
				Robot.M_StartRobotAbsMove(
					GetBox       := _toGet,
					UseClampA    := TRUE,
					UseClampB    := FALSE,
					Area         := Area,
					ClampA_Address := Address_A,
					ClampB_Address := 0,
					BoxReady_1   := tonBoxArriveDelay.Q OR BoxReady_1st,
					BoxReady_2   := FALSE);
			ELSIF Area = E_RobotArea.ShippingCCDPos THEN
				BoxReady_1st := TRUE;
				Robot.M_StartRobotAbsMove(
					GetBox       := TRUE,
					UseClampA    := TRUE,
					UseClampB    := FALSE,
					Area         := Area,
					ClampA_Address := 0,
					ClampB_Address := 0,
					BoxReady_1   := BoxReady_1st,
					BoxReady_2   := FALSE);
			ELSIF Area = E_RobotArea.ShippingFeedOutEmptyBox THEN
				BoxReady_1st := TRUE;
				Robot.M_StartRobotAbsMove(
					GetBox       := _toGet,
					UseClampA    := TRUE,
					UseClampB    := FALSE,
					Area         := Area,
					ClampA_Address := Address_A,
					ClampB_Address := 0,
					BoxReady_1   := BoxReady_1st,
					BoxReady_2   := FALSE);
			ELSE
				IF Area = E_RobotArea.ShippingBufferArea AND NOT _toGet THEN
					// Buffer Put 已設好 BoxReady
				ELSIF Area = E_RobotArea.ShippingBufferArea AND _toGet THEN
					// Buffer Get 已設好 BoxReady
				ELSE
					BoxReady_1st := TRUE;
				END_IF
				Robot.M_StartRobotAbsMove(
					GetBox       := _toGet,
					UseClampA    := TRUE,
					UseClampB    := FALSE,
					Area         := Area,
					ClampA_Address := Address_A,
					ClampB_Address := 0,
					BoxReady_1   := BoxReady_1st,
					BoxReady_2   := FALSE);
			END_IF
			_bAbsMoveStarted := TRUE;	// 標記真的有送過 Start 命令
		ELSIF NOT _bAbsMoveStarted THEN
			// Done=TRUE 但從未送過 Start → stale 狀態（續做 / Phase 1 殘留）
			// 先清掉 robot 命令，等 Done 變 FALSE 才能進入正常流程，避免 ghost completion
			Robot.M_ResetRobotAbsMove(TRUE, FALSE);
		ELSE
			// 真的完成（Done 從 FALSE → TRUE）→ 轉 15100
			// 不做手臂 ClampA_Sensor 驗證 — 對齊 step 5000 ELSE,軌道 sensor 把關時機,PLC 信任 Done
			TON_RobotActionTimeOut.IN := FALSE;
			tonBoxArriveDelay.IN      := FALSE;
			_bAbsMoveStarted          := FALSE;
			uiExecutingStep := 15100;
		END_IF

		IF TON_RobotActionTimeOut.Q THEN
			uiResumeStep := 15000;
			strStatus := 'FB_ShippingRobotTransfer Step 15000: Robot AbsMove timeout';
			Status := strStatus;
			Error := TRUE;
			_Abort       := TRUE;
		END_IF
		IF Robot._DI1.Error THEN
			uiResumeStep := 15000;
			strStatus    := CONCAT('TO: Robot Error ', Robot.ErrMsg);
			Status := strStatus;
			Error := TRUE;
			_Abort       := TRUE;
		END_IF

	15100: // TO Reset Robot command
		Robot.M_ResetRobotAbsMove(TRUE, FALSE);
		TON_CheckRobotDoneTimeOut.IN := TRUE;
		IF NOT Robot._DI1.Done THEN
			TON_CheckRobotDoneTimeOut.IN := FALSE;
			uiExecutingStep := 20000;
		END_IF
		IF TON_CheckRobotDoneTimeOut.Q THEN
			uiResumeStep := 15100;
			strStatus := 'FB_ShippingRobotTransfer Step 15100: Robot Reset timeout';
			Status := strStatus;
			Error := TRUE;
			_Abort       := TRUE;
		END_IF
		IF Robot._DI1.Error THEN
			uiResumeStep := 15100;
			strStatus    := CONCAT('TO Reset: Robot Error ', Robot.ErrMsg);
			Status := strStatus;
			Error := TRUE;
			_Abort       := TRUE;
		END_IF

	// ============================================================
	// Phase 2 (TO): 區域後置作業
	// ============================================================
	20000: // TO 後置
		// TransmitCVEnd: 停止輸送帶 — Phase 2 SameSize 撤銷請求,DifferentSize 直接停
		IF _toArea = E_RobotArea.TransmitCV_End THEN
			bMoveConveyorForward  := FALSE;
			bMoveConveyorBackward := FALSE;
			IF bIsSameSize THEN
				IF __ISVALIDREF(SameSizeCVRequest) THEN
					SameSizeCVRequest.bShippingTransfer_NeedForward  := FALSE;
					SameSizeCVRequest.bShippingTransfer_NeedBackward := FALSE;
				END_IF
			ELSIF __ISVALIDREF(ConveyorMotor) THEN
				ConveyorMotor.M_MotorStop();
			END_IF
		END_IF

		// Left/Right: 檢查是否需要 buzz
		IF (_toArea = E_RobotArea.ShippingRobotLeft OR _toArea = E_RobotArea.ShippingRobotRight)
			AND bCompleteRequest THEN
			uiExecutingStep := 25000;
		ELSE
			uiExecutingStep := 98000;
		END_IF

	// ============================================================
	// Phase 3: 警報 (buzz/lamp 閃爍)
	// ============================================================
	25000: // Buzz + Lamp 閃爍
		BuzzBlinker(ENABLE := TRUE, TIMELOW := T#0.3S, TIMEHIGH := T#0.3S, OUT => Buzz);
		LightBlinker(ENABLE := TRUE, TIMELOW := T#0.3S, TIMEHIGH := T#0.3S, OUT => RedLamp);
		TrigBuzz(CLK := Buzz);
		TrigLight(CLK := RedLamp);
		IF TrigBuzz.Q THEN
			BlinkInfo.BuzzCount := BlinkInfo.BuzzCount + 1;
		END_IF
		IF TrigLight.Q THEN
			BlinkInfo.LightCount := BlinkInfo.LightCount + 1;
		END_IF

		IF BlinkInfo.BuzzCount >= BlinkInfo.MaxBuzzCOunt AND BlinkInfo.LightCount >= BlinkInfo.MaxLightCount THEN
			TON_BlinkDelay.IN := TRUE;
			IF TON_BlinkDelay.Q THEN
				uiExecutingStep := 98000;
			END_IF
		END_IF

	// ============================================================
	// 完成
	// ============================================================
	98000:	// 完成前驗證 — 機構靜止 + 警示輸出歸零後才允許進 99000
		// 主動下停止指令 — Phase 2 SameSize 撤銷請求,DifferentSize 直接停
		bMoveConveyorForward  := FALSE;
		bMoveConveyorBackward := FALSE;
		IF bIsSameSize THEN
			IF __ISVALIDREF(SameSizeCVRequest) THEN
				SameSizeCVRequest.bShippingTransfer_NeedForward  := FALSE;
				SameSizeCVRequest.bShippingTransfer_NeedBackward := FALSE;
			END_IF
		ELSIF __ISVALIDREF(ConveyorMotor) THEN
			ConveyorMotor.M_MotorStop();
		END_IF
		// 強制關 Buzz / RedLamp，避免 step 25000 離開時殘留 HIGH
		BuzzBlinker(ENABLE := FALSE, OUT => Buzz);
		LightBlinker(ENABLE := FALSE, OUT => RedLamp);
		Buzz    := FALSE;
		RedLamp := FALSE;

		// 等輸送帶真的停下來
		TON_MechTimeOut.IN := TRUE;
		IF NOT __ISVALIDREF(ConveyorMotor)
		   OR (NOT ConveyorMotor.InForWard AND NOT ConveyorMotor.InBackWard) THEN
			TON_MechTimeOut.IN := FALSE;
			uiExecutingStep := 99000;
		ELSIF TON_MechTimeOut.Q THEN
			uiResumeStep := 98000;
			strStatus := 'FB_ShippingRobotTransfer Step 98000: Conveyor settle timeout';
			Status    := strStatus;
			Error     := TRUE;
			_Abort    := TRUE;
		END_IF

	99000:
		// Timer 全清
		TON_BlinkDelay.IN            := FALSE;
		TON_MechTimeOut.IN           := FALSE;
		TON_ServiceWatchDog.IN       := FALSE;
		TON_RobotActionTimeOut.IN    := FALSE;
		TON_CheckRobotDoneTimeOut.IN := FALSE;
		tonBoxArriveDelay.IN         := FALSE;
		TON_RSR02HomingTimeOut.IN    := FALSE;

		// 警示旗標歸零
		BlinkInfo.BuzzCount  := 0;
		BlinkInfo.LightCount := 0;
		Buzz    := FALSE;
		RedLamp := FALSE;

		// 動作旗標歸零
		bMoveConveyorForward  := FALSE;
		bMoveConveyorBackward := FALSE;

		// 暫存狀態歸零，確保下次 Execute 從乾淨狀態開始
		BoxReady_1st     := FALSE;
		Address_A        := 0;
		uiGetStep        := 0;
		_bRetry          := FALSE;
		_bAbsMoveStarted := FALSE;
		bCompleteRequest := FALSE;

		Status    := 'FB_ShippingRobotTransfer Step 99000: Process completed';
		_Executed := TRUE;	// ★ 必須最後設，確保旗標已全部清乾淨才宣告 Done

END_CASE

// 狀態機切換
IF NOT Execute THEN
	IF uiExecutingStep > 0 AND uiExecutingStep < 99000 THEN
		// 動作進行中被拉低 Execute → 強制走 Abort 流程把 robot/conveyor/cylinder 收乾淨
		strStatus := 'FB_ShippingRobotTransfer: Execute deasserted mid-operation';
		Status    := strStatus;
		_Abort    := TRUE;
		eState    := STATE_ABORTING;
	ELSE
		eState := STATE_RESETTING;
	END_IF
ELSIF _Error THEN
	eState := STATE_ERROR;
ELSIF _Abort OR Abort THEN
	eState := STATE_ABORTING;
ELSIF _Executed THEN
	eState := STATE_DONE;
END_IF
END_METHOD

METHOD M_STATE_HELD
VAR_INPUT
END_VAR
Busy   := FALSE;
Paused := TRUE;

CASE uiHeldStep OF
	0:
		uiHeldStep := 9999;
	9999:
		_HeldCompleted := TRUE;
END_CASE

IF _HeldCompleted AND NOT Pause THEN
	eState := STATE_UnHold;
END_IF
END_METHOD

METHOD M_STATE_HOLDING
VAR_INPUT
END_VAR
CASE uiHoldingStep OF
	0:
		// Pause 期間把所有計時器停掉，避免 watchdog 在暫停時跑滿後 resume 立刻誤觸發 Abort
		TON_RobotActionTimeOut.IN    := FALSE;
		TON_CheckRobotDoneTimeOut.IN := FALSE;
		TON_MechTimeOut.IN           := FALSE;
		TON_ServiceWatchDog.IN       := FALSE;
		tonBoxArriveDelay.IN         := FALSE;
		uiHoldingStep := 9999;
	9999:
		_HoldingCompleted := TRUE;
END_CASE

IF _HoldingCompleted THEN
	eState := STATE_Held;
END_IF
END_METHOD

METHOD M_STATE_RESETTING
VAR_INPUT
END_VAR
// Done := false 更改到Dormant 清除確保，上位檢查到done 後可以直接下Execute

CASE uiResettingStep OF
	0:
		bCompleteRequest := FALSE;
		bMoveConveyorForward  := FALSE;
		bMoveConveyorBackward := FALSE;
		_bAbsMoveStarted := FALSE;	// 雙保險:RESETTING → DORMANT 路徑,確保 stale ghost-completion flag 不殘留
		TON_RobotActionTimeOut.IN    := FALSE;
		TON_CheckRobotDoneTimeOut.IN := FALSE;
		TON_BlinkDelay.IN            := FALSE;
		TON_RSR02HomingTimeOut.IN    := FALSE;

		// 停止輸送帶 — Phase 2:DifferentSide 直接停;SameSide 撤銷請求 (arbiter 看到沒人 request 會自動停)
		Motor.List.TransmitDifferentSideCV.M_MotorStop();
		IF __ISVALIDREF(SameSizeCVRequest) THEN
			SameSizeCVRequest.bShippingTransfer_NeedForward  := FALSE;
			SameSizeCVRequest.bShippingTransfer_NeedBackward := FALSE;
		END_IF
		uiResettingStep := 200;

	200:
		// 等氣缸縮回 (如果有的話)
		IF NOT __ISVALIDREF(Cylinder) OR Cylinder.List.fbShippingBuffer_Press.InRearPosition THEN
			uiResettingStep := 300;
		ELSE
			Cylinder.List.fbShippingBuffer_Press.M_Retract();
		END_IF

	300:

		Robot.M_ResetAllCommand();
		IF Robot.M_CheckResetAllCommand() THEN
			uiResettingStep := 9999;
		END_IF

	9999:
		_ResetCompleted := TRUE;
END_CASE

IF _ResetCompleted THEN
	eState := STATE_DORMANT;
END_IF
END_METHOD

METHOD M_STATE_UNHOLD
VAR_INPUT
END_VAR
CASE uiUnholdStep OF
	0:
		uiUnholdStep := 9999;
	9999:
		_UnholdCompleted := TRUE;
END_CASE

IF _UnholdCompleted THEN
	Paused := FALSE;
	eState := STATE_EXECUTING;
END_IF
END_METHOD

END_FUNCTION_BLOCK

// ---- Library/20_MachineUnits/22_AllocateArea/Service/FB_SameSizeCV_ReverseBoxToWareHouse.TcPOU
// FB_SameSizeCV_ReverseBoxToWareHouse
// 同尺寸軌道逆向送盒入倉/NG 服務
// 流程: 擋盒 SM (Press3 後壓 + Press4 擋第二盒, ref AllocatedConveyor) → 軌道送到 NearStorage → 大手臂取盒 → 入倉 or NG區
// 支援: 單爪A / 單爪B / 雙爪 (2盒連續)
//
// 狀態機架構: FB_ObjectBase_V2 + IBasicElement
//   DORMANT → EXECUTING → DONE / ABORTING → ABORTED → RESETTING → DORMANT

FUNCTION_BLOCK FB_SameSizeCV_ReverseBoxToWareHouse EXTENDS FB_ObjectBase_V2 IMPLEMENTS IBasicElement

VAR_INPUT
	// ===== 盒子資訊 (由上層 FB 設定) =====
	bBoxA_Enable		: BOOL;						// A爪有盒子要處理
	eBoxA_Destination	: E_ReverseBoxDestination;	// A爪目的地: WareHouse / PullOut / NGConveyor
	iBoxA_Warehouse		: INT;						// (僅 Destination=WareHouse) 倉 (E_WareHouse: 1=A, 2=B)
	iBoxA_Level			: INT;						// (僅 Destination=WareHouse) 層 (1~10)
	iBoxA_Track			: INT;						// (僅 Destination=WareHouse) 軌 (1~20)
	iBoxA_PullOutSide	: INT;						// (僅 Destination=PullOut) 1=I3_Slide 左 / 2=I4_Slide 右

	bBoxB_Enable		: BOOL;						// B爪有盒子要處理 (FALSE=單爪)
	eBoxB_Destination	: E_ReverseBoxDestination;
	iBoxB_Warehouse		: INT;
	iBoxB_Level			: INT;
	iBoxB_Track			: INT;
	iBoxB_PullOutSide	: INT;						// 1=I3_Slide 左 / 2=I4_Slide 右

	NGAreaPosition		: INT := 3;					// NG 區 InOutConveyor Position
	PickupPosition		: INT := 2;					// 同尺寸輸送帶 為 2

	// ===== 硬體 REFERENCE =====
	Cylinder			: REFERENCE TO UNI_CylinderList;
	Motor				: REFERENCE TO UNI_MotorList;
	SameSizeCVRequest	: REFERENCE TO ST_SameSizeCVRequest;	// Phase 2 仲裁:本 FB 寫 bWareHouse_NeedBackward / bWareHouse_HoldStill
	Input				: ST_InputTable;
	OutPut				: ST_OutputTable;
	StorageRobot		: REFERENCE TO FB_FanucRobot_Basic_V2;
	WareHouse			: REFERENCE TO FB_WareHouse;
	PullOutConveyor		: REFERENCE TO FB_PullOutConveyorAction;	// PullOut 目的地需要

	Stop				: BOOL;
END_VAR

VAR_OUTPUT
	bBoxA_Done			: BOOL;				// A爪搬運完成 (入倉/PullOut/NG 三路皆算完成)
	bBoxB_Done			: BOOL;				// B爪搬運完成
END_VAR

VAR
	strStatus			: STRING;
	_UniqueErrorCode	: STRING;
	_bRetry				: BOOL;

	bDualGrip			: BOOL;
	bFirstClampIsA		: BOOL;
	bBoxReady			: BOOL;
	stWareHouseCoord	: ST_WareHouseCoordinates;

	// Timers
	TON_TimeOut			: TON;
	TON_ConveyorTimeOut	: TON;
	TON_RobotResetTimeOut : TON;
	TON_ArrivedDelay	: TON;
	tonDelay_SameSizeGetBox		: TON;	// 擋盒 SM:Detect6 50ms debounce (ref FB_RobotRegionMove_AllocatedConveyor)
	tonDelay_SameSizeDelayBox	: TON;	// 擋盒 SM:NearStorageSensor 1.5s 穩定確認

	// 擋盒 sub state (Phase 1/3 step 1100/3100 共用) — ref AllocatedConveyor uiSameGetBoxStep 0/100/200/300/400 pattern
	uiSameGetBoxStep	: UINT;

	// Resume
	uiResumeStep		: UDINT := 0;

	// Region move helpers
	NGRegionMove		: FB_RobotRegionMove_FeedInConveyor_V2;		// NG 目的地用 (InOutConveyor Pos 3)
	PullOutRegionMove	: FB_RobotRegionMove_PullOutConveyor;		// PullOut 目的地用 (新加)

	// STATE_ERROR retry framework (對齊 FB_ShippingRobotTransfer)
	trigErrorReset		: R_TRIG;
	tonErrorResetDelay	: TON;
	bErrorBlinking		: BOOL;

	// Phase 2:本 FB 有兩個 instance (Direct 在 FB_AllocateAreaWithRoundbelt + Orchestrator 在 FB_SameSizeCV_ReverseBatchPickAndPhoto)
	// shared SameSizeCVRequest flag 不能被 idle instance stomp。Step 寫 local intent,A00 + Busy gate 才 propagate。
	bIntent_NeedBackward	: BOOL;
	bIntent_HoldStill		: BOOL;
END_VAR

SUPER^.A10_StateControl();
A00_BasicUnits();

ACTION A00_BasicUnits:
TON_TimeOut(PT := T#60S);
TON_ConveyorTimeOut(PT := T#60S);
TON_RobotResetTimeOut(PT := T#30S);
TON_ArrivedDelay(PT:= T#300MS);
tonDelay_SameSizeGetBox(PT := T#50MS);
tonDelay_SameSizeDelayBox(PT := T#1500MS);

// Phase 2:Busy 期間才 propagate local intent 到 shared request flag,避免 idle instance stomp 別人的請求
IF Busy AND __ISVALIDREF(SameSizeCVRequest) THEN
	SameSizeCVRequest.bWareHouse_NeedBackward := bIntent_NeedBackward;
	SameSizeCVRequest.bWareHouse_HoldStill    := bIntent_HoldStill;
END_IF

NGRegionMove(
	Execute:= ,
	Abort:= ,
	Reset:= ,
	ObjectName:= ,
	Busy=> ,
	Done=> ,
	Aborted=> ,
	Error=> ,
	ErrorID=> ,
	Status=> ,
	UniqueErrorCode=> ,
	Robot:= StorageRobot,
	LowerConveyor:= Motor.List.LowCV,
	Input:= input,
	Info:= ,
	Stop:= );

PullOutRegionMove(
	Robot:= StorageRobot,
	PullOutConveyor:= PullOutConveyor,
	Stop:= Stop);
END_ACTION

